// TIA Portal V17 export
// export: Created 2025-03-05T08:03:03.6083882Z, ExportSetting WithDefaults, DisplayName Totally Integrated Automation Portal, DisplayVersion V17 Update 8, DisplayName TIA Portal Openness, DisplayVersion V17 Update 8, DisplayName TIA Portal Version Control Interface, DisplayVersion V17, DisplayName SINAMICS Startdrive Advanced, DisplayVersion V17 SP2, DisplayName SINAMICS Startdrive G110M, G120, G120C, G120D, G120P, G115D, DisplayVersion V17 SP2, DisplayName SINAMICS Startdrive G130, G150, S120, S150, SINAMICS MV, S210, DisplayVersion V17 SP2, DisplayName STEP 7 Professional, DisplayVersion V17 Update 8, DisplayName SINUMERIK ONE STEP 7 Toolbox, DisplayVersion V17 Update 12, DisplayName SINUMERIK 840D sl STEP 7 Toolbox, DisplayVersion V17 Update 12, DisplayName STEP 7 Safety, DisplayVersion V17 Update 6, DisplayName WinCC Advanced, DisplayVersion V17 Update 8
FUNCTION_BLOCK "FB21014_POWDER_FEEDER_PROFINET"   // FB21014, LAD
TITLE = FB21014 POWDER FEEDER PROFINET
{ S7_Optimized_Access := 'FALSE' }
VERSION : 0.1
// stored: AutoNumber false, IsIECCheckEnabled false, SetENOAutomatically false, UDAEnableTagReadback false
   VAR_INPUT
      "iHMI_Values Setpoints" : "POWDER FEEDER HMI VALUES SETPOINTS";
      "iHMI_Offsets Alarms and Warnings" : "POWDER FEEDER HMI OFFSETS ALARMS WARNINGS";
      "iCNC_Values Setpoints" : "POWDER FEEDER CNC VALUES SETPOINTS";
      iSTOP_LINE_1_VALUES_SETPOINTS : Struct
         LINE_1_GAS_FLOW : Real;   // LINE 1 GAS FLOW SETPOINT
         LINE_1_DISK_SPEED : Real;   // LINE 1 DISK SPEED SETPOINT
      END_STRUCT;
      iSTOP_LINE_2_VALUES_SETPOINTS : Struct
         LINE_2_GAS_FLOW : Real;   // LINE 2 GAS FLOW SETPOINT
         LINE_2_DISK_SPEED : Real;   // LINE 2 DISK SPEED SETPOINT
      END_STRUCT;
      iSTART_LINE_1_VALUES_SETPOINTS : Struct
         LINE_1_GAS_FLOW : Real;   // LINE 1 GAS FLOW SETPOINT
         LINE_1_DISK_SPEED : Real;   // LINE 1 DISK SPEED SETPOINT
      END_STRUCT;
      iSTART_LINE_2_VALUES_SETPOINTS : Struct
         LINE_2_GAS_FLOW : Real;   // LINE 2 GAS FLOW SETPOINT
         LINE_2_DISK_SPEED : Real;   // LINE 2 DISK SPEED SETPOINT
      END_STRUCT;
      iArgon_Carrier_Gas_Selected : Bool;
      iNitro_Carrier_Gas_Selected : Bool;
      iHelium_Carrier_Gas_Selected : Bool;
      iArgon30_Carrier_Gas_Selected : Bool;
      iLINE_1_ON_SEQ_ON : Bool;
      iLINE_2_ON_SEQ_ON : Bool;
      iLINE_1_OFF_SEQ_ON : Bool;
      iLINE_2_OFF_SEQ_ON : Bool;
      iLINE_1_STOPPED : Bool;   // HOPPER LINE 1 STOPPPED
      iLINE_2_STOPPED : Bool;   // HOPPER LINE 2 STOPPPED
   END_VAR
   VAR_OUTPUT
      oPLC_Aux : "POWDER FEEDER PLC AUXILIAR";
      oSTATION_WARNINGS : Bool;
      oWARNING_PF_LINE_1_GRAVIMETRIC_MODE_SELECTED : Bool;
      oWARNING_PF_LINE_2_GRAVIMETRIC_MODE_SELECTED : Bool;
   END_VAR
   VAR_IN_OUT
      ioPowder_Feeder_Unit_In_Out : "POWDER FEEDER OERLIKON";
   END_VAR
   VAR DB_SPECIFIC
      INPUT_SETTINGS : Struct
         UNIT_NUMBER : Int;
         FEEDER_NUMBER : Int;
      END_STRUCT;
      AUX_MANUAL_GAS_LINE_1 : Bool;   // AUX MANUAL GAS LINE 1
      AUX_MANUAL_GAS_LINE_2 : Bool;   // AUX MANUAL GAS LINE 2
      AUX_MANUAL_DISK_LINE_1 : Bool;   // AUX MANUAL DISK LINE 1
      AUX_MANUAL_DISK_LINE_2 : Bool;   // AUX MANUAL DISK LINE 2
      swapped : Word;
   END_VAR
   VAR_TEMP
      HMI_INPUT_MAN_MODE : Bool;
      OPTIONS_ON : Bool;
      OPTIONS_OFF : Bool;
      "VOLUMETRIC/GRAVIMETRIC" : Bool;
      "¿SUSTITUIR_VAR_CNC?" : Real;
      Retval_Fill_R : Real;
      DB_NUMBER : DInt;
   END_VAR
   VAR_TEMP   // added for the SCL form of the ladder/FBD networks
      _w1 : Bool;
   END_VAR
BEGIN

NETWORK
TITLE = READ INSTANCE DB NUMBER
      L     DINO;
      +     10#800000;
      T     #DB_NUMBER;

REGION Network 2: HMI INPUT
   // With Hmi Input we allow for user manipulation of feeder operating parameters. If not, they get overriden by robot interlock.
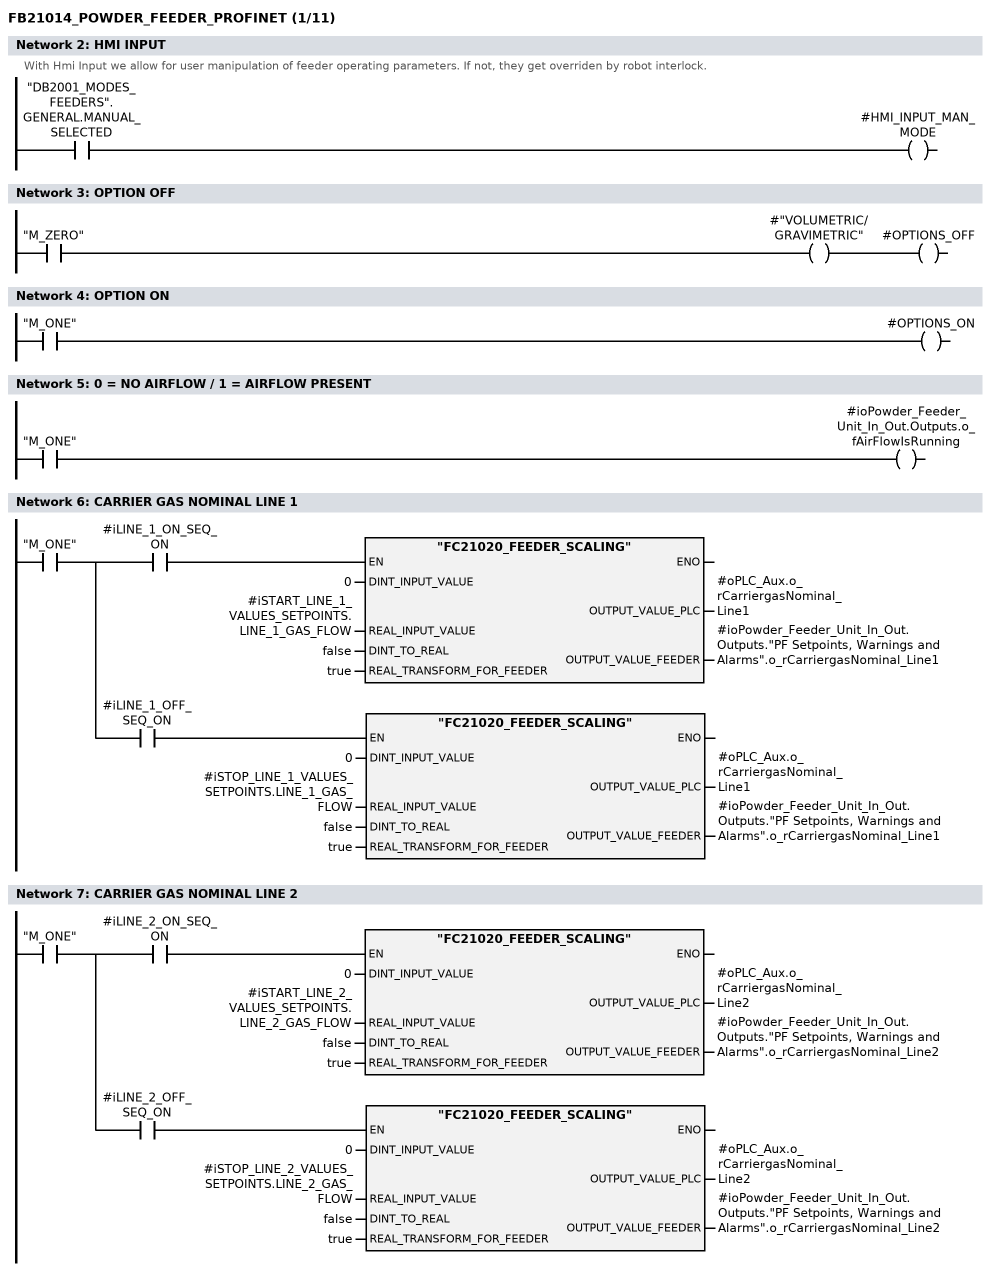
   RUNG wire#powerrail
      Contact( "DB2001_MODES_FEEDERS".GENERAL.MANUAL_SELECTED )
      Coil( #HMI_INPUT_MAN_MODE )
   END_RUNG
   // the same network as SCL:
   #HMI_INPUT_MAN_MODE := "DB2001_MODES_FEEDERS".GENERAL.MANUAL_SELECTED;
END_REGION

REGION Network 3: OPTION OFF
   RUNG wire#powerrail
      Contact( "M_ZERO" )
      Coil( #"VOLUMETRIC/GRAVIMETRIC" )
      Coil( #OPTIONS_OFF )
   END_RUNG
   // the same network as SCL:
   #"VOLUMETRIC/GRAVIMETRIC" := "M_ZERO";
   #OPTIONS_OFF := "M_ZERO";
END_REGION

REGION Network 4: OPTION ON
   RUNG wire#powerrail
      Contact( "M_ONE" )
      Coil( #OPTIONS_ON )
   END_RUNG
   // the same network as SCL:
   #OPTIONS_ON := "M_ONE";
END_REGION

REGION Network 5: 0 = NO AIRFLOW / 1 = AIRFLOW PRESENT
   RUNG wire#powerrail
      Contact( "M_ONE" )
      Coil( #ioPowder_Feeder_Unit_In_Out.Outputs.o_fAirFlowIsRunning )
   END_RUNG
   // the same network as SCL:
   #ioPowder_Feeder_Unit_In_Out.Outputs.o_fAirFlowIsRunning := "M_ONE";
END_REGION

REGION Network 6: CARRIER GAS NOMINAL LINE 1
   RUNG wire#powerrail
      Contact( "M_ONE" )
      wire#w1
      Contact( #iLINE_1_ON_SEQ_ON )
      "FC21020_FEEDER_SCALING"(DINT_INPUT_VALUE := 0, REAL_INPUT_VALUE := #iSTART_LINE_1_VALUES_SETPOINTS.LINE_1_GAS_FLOW, DINT_TO_REAL := false, REAL_TRANSFORM_FOR_FEEDER := true, OUTPUT_VALUE_PLC => #oPLC_Aux.o_rCarriergasNominal_Line1, OUTPUT_VALUE_FEEDER => #ioPowder_Feeder_Unit_In_Out.Outputs."PF Setpoints, Warnings and Alarms".o_rCarriergasNominal_Line1)
   END_RUNG
   RUNG wire#w1
      Contact( #iLINE_1_OFF_SEQ_ON )
      "FC21020_FEEDER_SCALING"(DINT_INPUT_VALUE := 0, REAL_INPUT_VALUE := #iSTOP_LINE_1_VALUES_SETPOINTS.LINE_1_GAS_FLOW, DINT_TO_REAL := false, REAL_TRANSFORM_FOR_FEEDER := true, OUTPUT_VALUE_PLC => #oPLC_Aux.o_rCarriergasNominal_Line1, OUTPUT_VALUE_FEEDER => #ioPowder_Feeder_Unit_In_Out.Outputs."PF Setpoints, Warnings and Alarms".o_rCarriergasNominal_Line1)
   END_RUNG
   // the same network as SCL:
   #_w1 := "M_ONE";
   IF "M_ONE" AND #iLINE_1_ON_SEQ_ON THEN
       "FC21020_FEEDER_SCALING"(DINT_INPUT_VALUE := 0,
                               REAL_INPUT_VALUE := #iSTART_LINE_1_VALUES_SETPOINTS.LINE_1_GAS_FLOW,
                               DINT_TO_REAL := false,
                               REAL_TRANSFORM_FOR_FEEDER := true,
                               OUTPUT_VALUE_PLC => #oPLC_Aux.o_rCarriergasNominal_Line1,
                               OUTPUT_VALUE_FEEDER => #ioPowder_Feeder_Unit_In_Out.Outputs."PF Setpoints, Warnings and Alarms".o_rCarriergasNominal_Line1);
   END_IF;
   IF #_w1 AND #iLINE_1_OFF_SEQ_ON THEN
       "FC21020_FEEDER_SCALING"(DINT_INPUT_VALUE := 0,
                               REAL_INPUT_VALUE := #iSTOP_LINE_1_VALUES_SETPOINTS.LINE_1_GAS_FLOW,
                               DINT_TO_REAL := false,
                               REAL_TRANSFORM_FOR_FEEDER := true,
                               OUTPUT_VALUE_PLC => #oPLC_Aux.o_rCarriergasNominal_Line1,
                               OUTPUT_VALUE_FEEDER => #ioPowder_Feeder_Unit_In_Out.Outputs."PF Setpoints, Warnings and Alarms".o_rCarriergasNominal_Line1);
   END_IF;
END_REGION

REGION Network 7: CARRIER GAS NOMINAL LINE 2
   RUNG wire#powerrail
      Contact( "M_ONE" )
      wire#w1
      Contact( #iLINE_2_ON_SEQ_ON )
      "FC21020_FEEDER_SCALING"(DINT_INPUT_VALUE := 0, REAL_INPUT_VALUE := #iSTART_LINE_2_VALUES_SETPOINTS.LINE_2_GAS_FLOW, DINT_TO_REAL := false, REAL_TRANSFORM_FOR_FEEDER := true, OUTPUT_VALUE_PLC => #oPLC_Aux.o_rCarriergasNominal_Line2, OUTPUT_VALUE_FEEDER => #ioPowder_Feeder_Unit_In_Out.Outputs."PF Setpoints, Warnings and Alarms".o_rCarriergasNominal_Line2)
   END_RUNG
   RUNG wire#w1
      Contact( #iLINE_2_OFF_SEQ_ON )
      "FC21020_FEEDER_SCALING"(DINT_INPUT_VALUE := 0, REAL_INPUT_VALUE := #iSTOP_LINE_2_VALUES_SETPOINTS.LINE_2_GAS_FLOW, DINT_TO_REAL := false, REAL_TRANSFORM_FOR_FEEDER := true, OUTPUT_VALUE_PLC => #oPLC_Aux.o_rCarriergasNominal_Line2, OUTPUT_VALUE_FEEDER => #ioPowder_Feeder_Unit_In_Out.Outputs."PF Setpoints, Warnings and Alarms".o_rCarriergasNominal_Line2)
   END_RUNG
   // the same network as SCL:
   #_w1 := "M_ONE";
   IF "M_ONE" AND #iLINE_2_ON_SEQ_ON THEN
       "FC21020_FEEDER_SCALING"(DINT_INPUT_VALUE := 0,
                               REAL_INPUT_VALUE := #iSTART_LINE_2_VALUES_SETPOINTS.LINE_2_GAS_FLOW,
                               DINT_TO_REAL := false,
                               REAL_TRANSFORM_FOR_FEEDER := true,
                               OUTPUT_VALUE_PLC => #oPLC_Aux.o_rCarriergasNominal_Line2,
                               OUTPUT_VALUE_FEEDER => #ioPowder_Feeder_Unit_In_Out.Outputs."PF Setpoints, Warnings and Alarms".o_rCarriergasNominal_Line2);
   END_IF;
   IF #_w1 AND #iLINE_2_OFF_SEQ_ON THEN
       "FC21020_FEEDER_SCALING"(DINT_INPUT_VALUE := 0,
                               REAL_INPUT_VALUE := #iSTOP_LINE_2_VALUES_SETPOINTS.LINE_2_GAS_FLOW,
                               DINT_TO_REAL := false,
                               REAL_TRANSFORM_FOR_FEEDER := true,
                               OUTPUT_VALUE_PLC => #oPLC_Aux.o_rCarriergasNominal_Line2,
                               OUTPUT_VALUE_FEEDER => #ioPowder_Feeder_Unit_In_Out.Outputs."PF Setpoints, Warnings and Alarms".o_rCarriergasNominal_Line2);
   END_IF;
END_REGION

REGION Network 8: DISK SPEED NOMINAL LINE 1
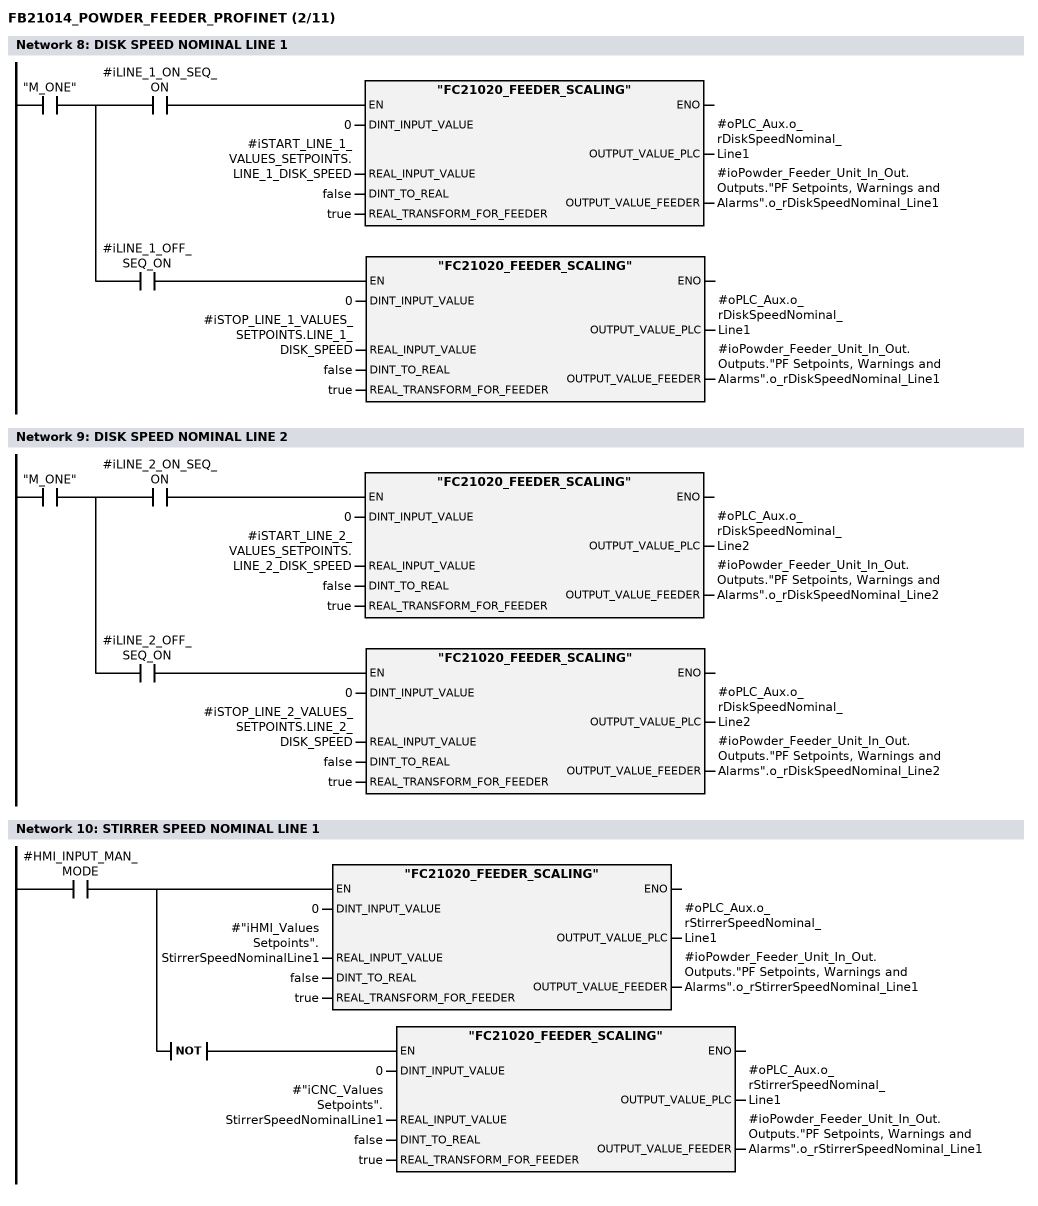
   RUNG wire#powerrail
      Contact( "M_ONE" )
      wire#w1
      Contact( #iLINE_1_ON_SEQ_ON )
      "FC21020_FEEDER_SCALING"(DINT_INPUT_VALUE := 0, REAL_INPUT_VALUE := #iSTART_LINE_1_VALUES_SETPOINTS.LINE_1_DISK_SPEED, DINT_TO_REAL := false, REAL_TRANSFORM_FOR_FEEDER := true, OUTPUT_VALUE_PLC => #oPLC_Aux.o_rDiskSpeedNominal_Line1, OUTPUT_VALUE_FEEDER => #ioPowder_Feeder_Unit_In_Out.Outputs."PF Setpoints, Warnings and Alarms".o_rDiskSpeedNominal_Line1)
   END_RUNG
   RUNG wire#w1
      Contact( #iLINE_1_OFF_SEQ_ON )
      "FC21020_FEEDER_SCALING"(DINT_INPUT_VALUE := 0, REAL_INPUT_VALUE := #iSTOP_LINE_1_VALUES_SETPOINTS.LINE_1_DISK_SPEED, DINT_TO_REAL := false, REAL_TRANSFORM_FOR_FEEDER := true, OUTPUT_VALUE_PLC => #oPLC_Aux.o_rDiskSpeedNominal_Line1, OUTPUT_VALUE_FEEDER => #ioPowder_Feeder_Unit_In_Out.Outputs."PF Setpoints, Warnings and Alarms".o_rDiskSpeedNominal_Line1)
   END_RUNG
   // the same network as SCL:
   #_w1 := "M_ONE";
   IF "M_ONE" AND #iLINE_1_ON_SEQ_ON THEN
       "FC21020_FEEDER_SCALING"(DINT_INPUT_VALUE := 0,
                               REAL_INPUT_VALUE := #iSTART_LINE_1_VALUES_SETPOINTS.LINE_1_DISK_SPEED,
                               DINT_TO_REAL := false,
                               REAL_TRANSFORM_FOR_FEEDER := true,
                               OUTPUT_VALUE_PLC => #oPLC_Aux.o_rDiskSpeedNominal_Line1,
                               OUTPUT_VALUE_FEEDER => #ioPowder_Feeder_Unit_In_Out.Outputs."PF Setpoints, Warnings and Alarms".o_rDiskSpeedNominal_Line1);
   END_IF;
   IF #_w1 AND #iLINE_1_OFF_SEQ_ON THEN
       "FC21020_FEEDER_SCALING"(DINT_INPUT_VALUE := 0,
                               REAL_INPUT_VALUE := #iSTOP_LINE_1_VALUES_SETPOINTS.LINE_1_DISK_SPEED,
                               DINT_TO_REAL := false,
                               REAL_TRANSFORM_FOR_FEEDER := true,
                               OUTPUT_VALUE_PLC => #oPLC_Aux.o_rDiskSpeedNominal_Line1,
                               OUTPUT_VALUE_FEEDER => #ioPowder_Feeder_Unit_In_Out.Outputs."PF Setpoints, Warnings and Alarms".o_rDiskSpeedNominal_Line1);
   END_IF;
END_REGION

REGION Network 9: DISK SPEED NOMINAL LINE 2
   RUNG wire#powerrail
      Contact( "M_ONE" )
      wire#w1
      Contact( #iLINE_2_ON_SEQ_ON )
      "FC21020_FEEDER_SCALING"(DINT_INPUT_VALUE := 0, REAL_INPUT_VALUE := #iSTART_LINE_2_VALUES_SETPOINTS.LINE_2_DISK_SPEED, DINT_TO_REAL := false, REAL_TRANSFORM_FOR_FEEDER := true, OUTPUT_VALUE_PLC => #oPLC_Aux.o_rDiskSpeedNominal_Line2, OUTPUT_VALUE_FEEDER => #ioPowder_Feeder_Unit_In_Out.Outputs."PF Setpoints, Warnings and Alarms".o_rDiskSpeedNominal_Line2)
   END_RUNG
   RUNG wire#w1
      Contact( #iLINE_2_OFF_SEQ_ON )
      "FC21020_FEEDER_SCALING"(DINT_INPUT_VALUE := 0, REAL_INPUT_VALUE := #iSTOP_LINE_2_VALUES_SETPOINTS.LINE_2_DISK_SPEED, DINT_TO_REAL := false, REAL_TRANSFORM_FOR_FEEDER := true, OUTPUT_VALUE_PLC => #oPLC_Aux.o_rDiskSpeedNominal_Line2, OUTPUT_VALUE_FEEDER => #ioPowder_Feeder_Unit_In_Out.Outputs."PF Setpoints, Warnings and Alarms".o_rDiskSpeedNominal_Line2)
   END_RUNG
   // the same network as SCL:
   #_w1 := "M_ONE";
   IF "M_ONE" AND #iLINE_2_ON_SEQ_ON THEN
       "FC21020_FEEDER_SCALING"(DINT_INPUT_VALUE := 0,
                               REAL_INPUT_VALUE := #iSTART_LINE_2_VALUES_SETPOINTS.LINE_2_DISK_SPEED,
                               DINT_TO_REAL := false,
                               REAL_TRANSFORM_FOR_FEEDER := true,
                               OUTPUT_VALUE_PLC => #oPLC_Aux.o_rDiskSpeedNominal_Line2,
                               OUTPUT_VALUE_FEEDER => #ioPowder_Feeder_Unit_In_Out.Outputs."PF Setpoints, Warnings and Alarms".o_rDiskSpeedNominal_Line2);
   END_IF;
   IF #_w1 AND #iLINE_2_OFF_SEQ_ON THEN
       "FC21020_FEEDER_SCALING"(DINT_INPUT_VALUE := 0,
                               REAL_INPUT_VALUE := #iSTOP_LINE_2_VALUES_SETPOINTS.LINE_2_DISK_SPEED,
                               DINT_TO_REAL := false,
                               REAL_TRANSFORM_FOR_FEEDER := true,
                               OUTPUT_VALUE_PLC => #oPLC_Aux.o_rDiskSpeedNominal_Line2,
                               OUTPUT_VALUE_FEEDER => #ioPowder_Feeder_Unit_In_Out.Outputs."PF Setpoints, Warnings and Alarms".o_rDiskSpeedNominal_Line2);
   END_IF;
END_REGION

REGION Network 10: STIRRER SPEED NOMINAL LINE 1
   RUNG wire#powerrail
      Contact( #HMI_INPUT_MAN_MODE )
      wire#w1
      "FC21020_FEEDER_SCALING"(DINT_INPUT_VALUE := 0, REAL_INPUT_VALUE := #"iHMI_Values Setpoints".StirrerSpeedNominalLine1, DINT_TO_REAL := false, REAL_TRANSFORM_FOR_FEEDER := true, OUTPUT_VALUE_PLC => #oPLC_Aux.o_rStirrerSpeedNominal_Line1, OUTPUT_VALUE_FEEDER => #ioPowder_Feeder_Unit_In_Out.Outputs."PF Setpoints, Warnings and Alarms".o_rStirrerSpeedNominal_Line1)
   END_RUNG
   RUNG wire#w1
      Not()
      "FC21020_FEEDER_SCALING"(DINT_INPUT_VALUE := 0, REAL_INPUT_VALUE := #"iCNC_Values Setpoints".StirrerSpeedNominalLine1, DINT_TO_REAL := false, REAL_TRANSFORM_FOR_FEEDER := true, OUTPUT_VALUE_PLC => #oPLC_Aux.o_rStirrerSpeedNominal_Line1, OUTPUT_VALUE_FEEDER => #ioPowder_Feeder_Unit_In_Out.Outputs."PF Setpoints, Warnings and Alarms".o_rStirrerSpeedNominal_Line1)
   END_RUNG
   // the same network as SCL:
   IF #HMI_INPUT_MAN_MODE THEN
       "FC21020_FEEDER_SCALING"(DINT_INPUT_VALUE := 0,
                               REAL_INPUT_VALUE := #"iHMI_Values Setpoints".StirrerSpeedNominalLine1,
                               DINT_TO_REAL := false,
                               REAL_TRANSFORM_FOR_FEEDER := true,
                               OUTPUT_VALUE_PLC => #oPLC_Aux.o_rStirrerSpeedNominal_Line1,
                               OUTPUT_VALUE_FEEDER => #ioPowder_Feeder_Unit_In_Out.Outputs."PF Setpoints, Warnings and Alarms".o_rStirrerSpeedNominal_Line1);
   END_IF;
   IF NOT #HMI_INPUT_MAN_MODE THEN
       "FC21020_FEEDER_SCALING"(DINT_INPUT_VALUE := 0,
                               REAL_INPUT_VALUE := #"iCNC_Values Setpoints".StirrerSpeedNominalLine1,
                               DINT_TO_REAL := false,
                               REAL_TRANSFORM_FOR_FEEDER := true,
                               OUTPUT_VALUE_PLC => #oPLC_Aux.o_rStirrerSpeedNominal_Line1,
                               OUTPUT_VALUE_FEEDER => #ioPowder_Feeder_Unit_In_Out.Outputs."PF Setpoints, Warnings and Alarms".o_rStirrerSpeedNominal_Line1);
   END_IF;
END_REGION

REGION Network 11: STIRRER SPEED NOMINAL LINE 2
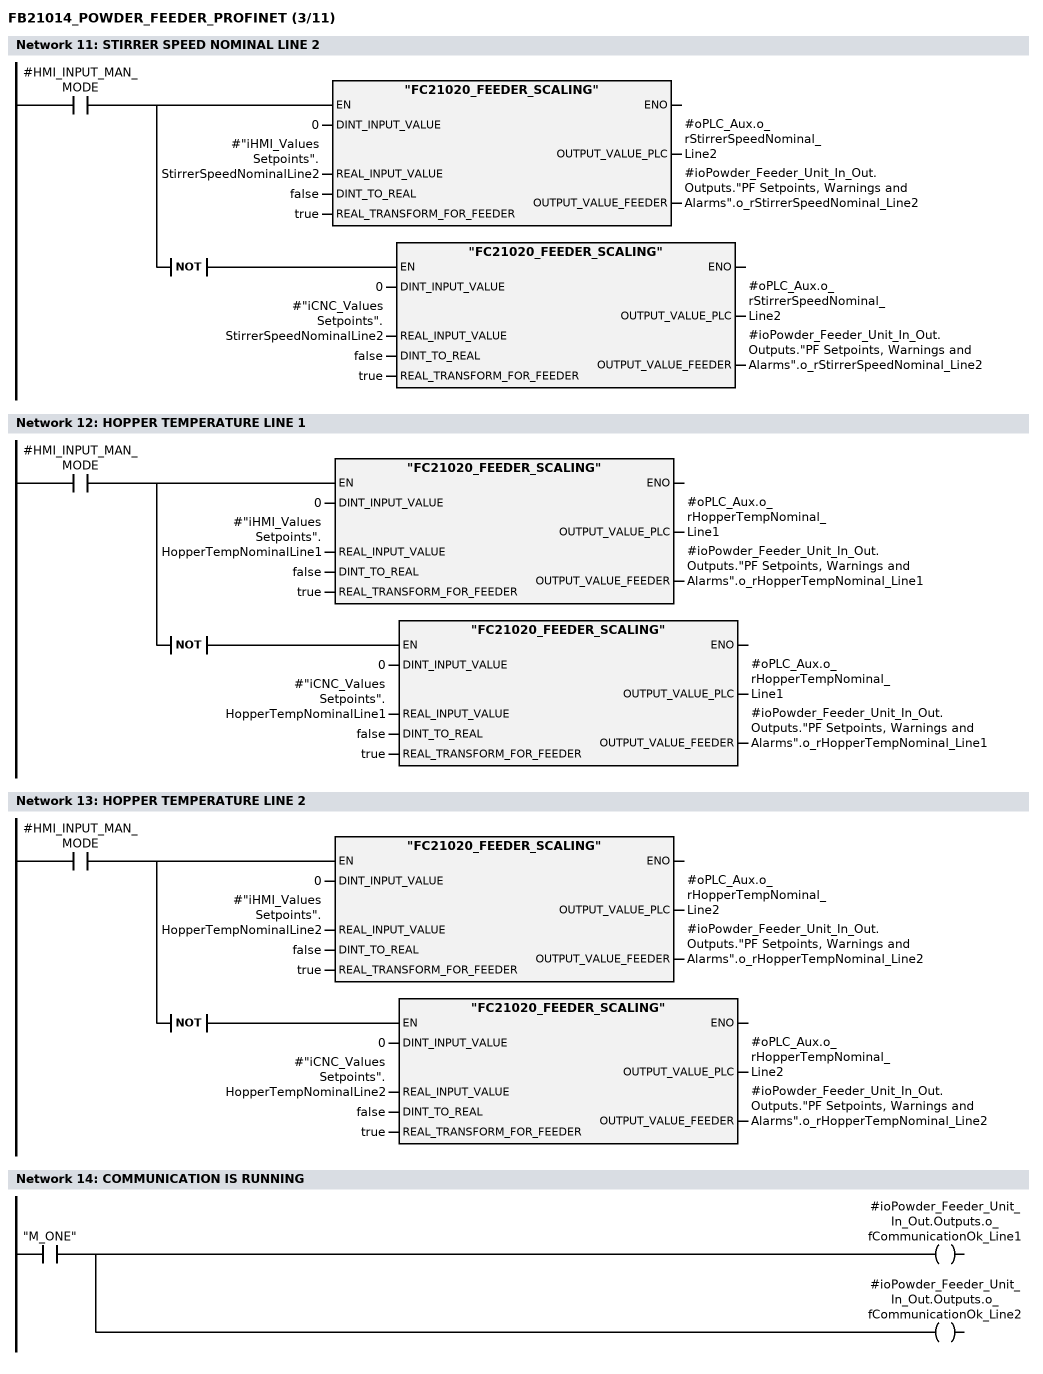
   RUNG wire#powerrail
      Contact( #HMI_INPUT_MAN_MODE )
      wire#w1
      "FC21020_FEEDER_SCALING"(DINT_INPUT_VALUE := 0, REAL_INPUT_VALUE := #"iHMI_Values Setpoints".StirrerSpeedNominalLine2, DINT_TO_REAL := false, REAL_TRANSFORM_FOR_FEEDER := true, OUTPUT_VALUE_PLC => #oPLC_Aux.o_rStirrerSpeedNominal_Line2, OUTPUT_VALUE_FEEDER => #ioPowder_Feeder_Unit_In_Out.Outputs."PF Setpoints, Warnings and Alarms".o_rStirrerSpeedNominal_Line2)
   END_RUNG
   RUNG wire#w1
      Not()
      "FC21020_FEEDER_SCALING"(DINT_INPUT_VALUE := 0, REAL_INPUT_VALUE := #"iCNC_Values Setpoints".StirrerSpeedNominalLine2, DINT_TO_REAL := false, REAL_TRANSFORM_FOR_FEEDER := true, OUTPUT_VALUE_PLC => #oPLC_Aux.o_rStirrerSpeedNominal_Line2, OUTPUT_VALUE_FEEDER => #ioPowder_Feeder_Unit_In_Out.Outputs."PF Setpoints, Warnings and Alarms".o_rStirrerSpeedNominal_Line2)
   END_RUNG
   // the same network as SCL:
   IF #HMI_INPUT_MAN_MODE THEN
       "FC21020_FEEDER_SCALING"(DINT_INPUT_VALUE := 0,
                               REAL_INPUT_VALUE := #"iHMI_Values Setpoints".StirrerSpeedNominalLine2,
                               DINT_TO_REAL := false,
                               REAL_TRANSFORM_FOR_FEEDER := true,
                               OUTPUT_VALUE_PLC => #oPLC_Aux.o_rStirrerSpeedNominal_Line2,
                               OUTPUT_VALUE_FEEDER => #ioPowder_Feeder_Unit_In_Out.Outputs."PF Setpoints, Warnings and Alarms".o_rStirrerSpeedNominal_Line2);
   END_IF;
   IF NOT #HMI_INPUT_MAN_MODE THEN
       "FC21020_FEEDER_SCALING"(DINT_INPUT_VALUE := 0,
                               REAL_INPUT_VALUE := #"iCNC_Values Setpoints".StirrerSpeedNominalLine2,
                               DINT_TO_REAL := false,
                               REAL_TRANSFORM_FOR_FEEDER := true,
                               OUTPUT_VALUE_PLC => #oPLC_Aux.o_rStirrerSpeedNominal_Line2,
                               OUTPUT_VALUE_FEEDER => #ioPowder_Feeder_Unit_In_Out.Outputs."PF Setpoints, Warnings and Alarms".o_rStirrerSpeedNominal_Line2);
   END_IF;
END_REGION

REGION Network 12: HOPPER TEMPERATURE LINE 1
   RUNG wire#powerrail
      Contact( #HMI_INPUT_MAN_MODE )
      wire#w1
      "FC21020_FEEDER_SCALING"(DINT_INPUT_VALUE := 0, REAL_INPUT_VALUE := #"iHMI_Values Setpoints".HopperTempNominalLine1, DINT_TO_REAL := false, REAL_TRANSFORM_FOR_FEEDER := true, OUTPUT_VALUE_PLC => #oPLC_Aux.o_rHopperTempNominal_Line1, OUTPUT_VALUE_FEEDER => #ioPowder_Feeder_Unit_In_Out.Outputs."PF Setpoints, Warnings and Alarms".o_rHopperTempNominal_Line1)
   END_RUNG
   RUNG wire#w1
      Not()
      "FC21020_FEEDER_SCALING"(DINT_INPUT_VALUE := 0, REAL_INPUT_VALUE := #"iCNC_Values Setpoints".HopperTempNominalLine1, DINT_TO_REAL := false, REAL_TRANSFORM_FOR_FEEDER := true, OUTPUT_VALUE_PLC => #oPLC_Aux.o_rHopperTempNominal_Line1, OUTPUT_VALUE_FEEDER => #ioPowder_Feeder_Unit_In_Out.Outputs."PF Setpoints, Warnings and Alarms".o_rHopperTempNominal_Line1)
   END_RUNG
   // the same network as SCL:
   IF #HMI_INPUT_MAN_MODE THEN
       "FC21020_FEEDER_SCALING"(DINT_INPUT_VALUE := 0,
                               REAL_INPUT_VALUE := #"iHMI_Values Setpoints".HopperTempNominalLine1,
                               DINT_TO_REAL := false,
                               REAL_TRANSFORM_FOR_FEEDER := true,
                               OUTPUT_VALUE_PLC => #oPLC_Aux.o_rHopperTempNominal_Line1,
                               OUTPUT_VALUE_FEEDER => #ioPowder_Feeder_Unit_In_Out.Outputs."PF Setpoints, Warnings and Alarms".o_rHopperTempNominal_Line1);
   END_IF;
   IF NOT #HMI_INPUT_MAN_MODE THEN
       "FC21020_FEEDER_SCALING"(DINT_INPUT_VALUE := 0,
                               REAL_INPUT_VALUE := #"iCNC_Values Setpoints".HopperTempNominalLine1,
                               DINT_TO_REAL := false,
                               REAL_TRANSFORM_FOR_FEEDER := true,
                               OUTPUT_VALUE_PLC => #oPLC_Aux.o_rHopperTempNominal_Line1,
                               OUTPUT_VALUE_FEEDER => #ioPowder_Feeder_Unit_In_Out.Outputs."PF Setpoints, Warnings and Alarms".o_rHopperTempNominal_Line1);
   END_IF;
END_REGION

REGION Network 13: HOPPER TEMPERATURE LINE 2
   RUNG wire#powerrail
      Contact( #HMI_INPUT_MAN_MODE )
      wire#w1
      "FC21020_FEEDER_SCALING"(DINT_INPUT_VALUE := 0, REAL_INPUT_VALUE := #"iHMI_Values Setpoints".HopperTempNominalLine2, DINT_TO_REAL := false, REAL_TRANSFORM_FOR_FEEDER := true, OUTPUT_VALUE_PLC => #oPLC_Aux.o_rHopperTempNominal_Line2, OUTPUT_VALUE_FEEDER => #ioPowder_Feeder_Unit_In_Out.Outputs."PF Setpoints, Warnings and Alarms".o_rHopperTempNominal_Line2)
   END_RUNG
   RUNG wire#w1
      Not()
      "FC21020_FEEDER_SCALING"(DINT_INPUT_VALUE := 0, REAL_INPUT_VALUE := #"iCNC_Values Setpoints".HopperTempNominalLine2, DINT_TO_REAL := false, REAL_TRANSFORM_FOR_FEEDER := true, OUTPUT_VALUE_PLC => #oPLC_Aux.o_rHopperTempNominal_Line2, OUTPUT_VALUE_FEEDER => #ioPowder_Feeder_Unit_In_Out.Outputs."PF Setpoints, Warnings and Alarms".o_rHopperTempNominal_Line2)
   END_RUNG
   // the same network as SCL:
   IF #HMI_INPUT_MAN_MODE THEN
       "FC21020_FEEDER_SCALING"(DINT_INPUT_VALUE := 0,
                               REAL_INPUT_VALUE := #"iHMI_Values Setpoints".HopperTempNominalLine2,
                               DINT_TO_REAL := false,
                               REAL_TRANSFORM_FOR_FEEDER := true,
                               OUTPUT_VALUE_PLC => #oPLC_Aux.o_rHopperTempNominal_Line2,
                               OUTPUT_VALUE_FEEDER => #ioPowder_Feeder_Unit_In_Out.Outputs."PF Setpoints, Warnings and Alarms".o_rHopperTempNominal_Line2);
   END_IF;
   IF NOT #HMI_INPUT_MAN_MODE THEN
       "FC21020_FEEDER_SCALING"(DINT_INPUT_VALUE := 0,
                               REAL_INPUT_VALUE := #"iCNC_Values Setpoints".HopperTempNominalLine2,
                               DINT_TO_REAL := false,
                               REAL_TRANSFORM_FOR_FEEDER := true,
                               OUTPUT_VALUE_PLC => #oPLC_Aux.o_rHopperTempNominal_Line2,
                               OUTPUT_VALUE_FEEDER => #ioPowder_Feeder_Unit_In_Out.Outputs."PF Setpoints, Warnings and Alarms".o_rHopperTempNominal_Line2);
   END_IF;
END_REGION

REGION Network 14: COMMUNICATION IS RUNNING
   RUNG wire#powerrail
      Contact( "M_ONE" )
      wire#w1
      Coil( #ioPowder_Feeder_Unit_In_Out.Outputs.o_fCommunicationOk_Line1 )
   END_RUNG
   RUNG wire#w1
      Coil( #ioPowder_Feeder_Unit_In_Out.Outputs.o_fCommunicationOk_Line2 )
   END_RUNG
   // the same network as SCL:
   #ioPowder_Feeder_Unit_In_Out.Outputs.o_fCommunicationOk_Line1 := "M_ONE";
   #ioPowder_Feeder_Unit_In_Out.Outputs.o_fCommunicationOk_Line2 := "M_ONE";
END_REGION

REGION Network 15: VOLUMETRIC MODE ON
   // Volumetric Mode On = 1 for Twin 150
   // Gravimetric Mode - n/a for Twin 150
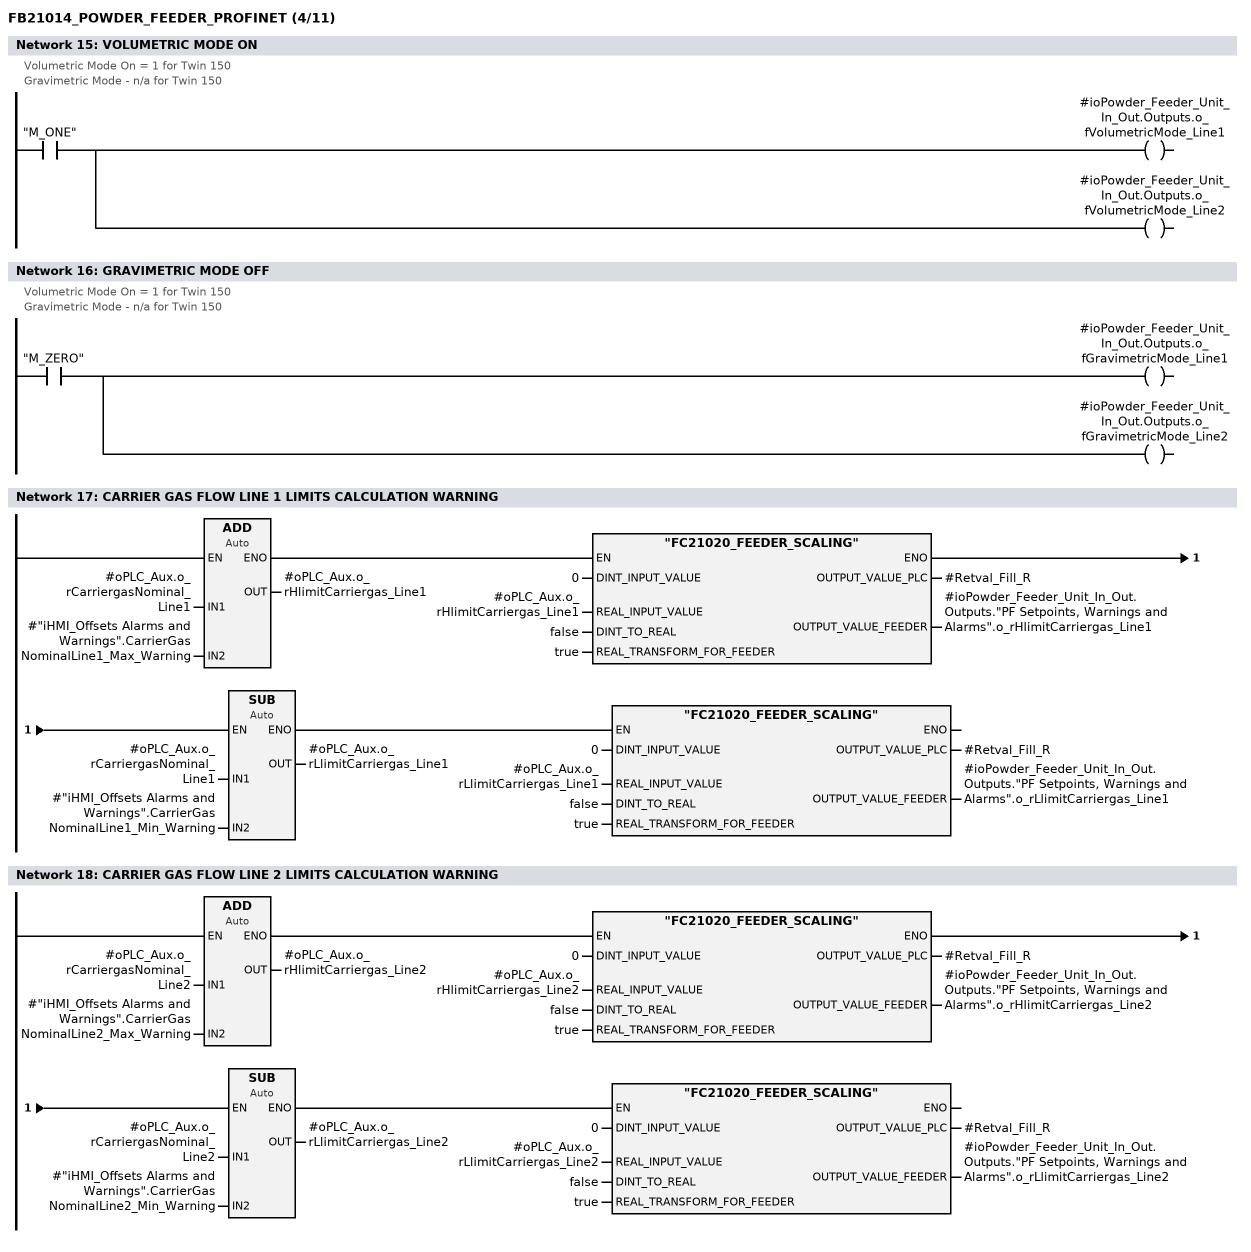
   RUNG wire#powerrail
      Contact( "M_ONE" )
      wire#w1
      Coil( #ioPowder_Feeder_Unit_In_Out.Outputs.o_fVolumetricMode_Line1 )
   END_RUNG
   RUNG wire#w1
      Coil( #ioPowder_Feeder_Unit_In_Out.Outputs.o_fVolumetricMode_Line2 )
   END_RUNG
   // the same network as SCL:
   #ioPowder_Feeder_Unit_In_Out.Outputs.o_fVolumetricMode_Line1 := "M_ONE";
   #ioPowder_Feeder_Unit_In_Out.Outputs.o_fVolumetricMode_Line2 := "M_ONE";
END_REGION

REGION Network 16: GRAVIMETRIC MODE OFF
   // Volumetric Mode On = 1 for Twin 150
   // Gravimetric Mode - n/a for Twin 150
   RUNG wire#powerrail
      Contact( "M_ZERO" )
      wire#w1
      Coil( #ioPowder_Feeder_Unit_In_Out.Outputs.o_fGravimetricMode_Line1 )
   END_RUNG
   RUNG wire#w1
      Coil( #ioPowder_Feeder_Unit_In_Out.Outputs.o_fGravimetricMode_Line2 )
   END_RUNG
   // the same network as SCL:
   #ioPowder_Feeder_Unit_In_Out.Outputs.o_fGravimetricMode_Line1 := "M_ZERO";
   #ioPowder_Feeder_Unit_In_Out.Outputs.o_fGravimetricMode_Line2 := "M_ZERO";
END_REGION

REGION Network 17: CARRIER GAS FLOW LINE 1 LIMITS CALCULATION WARNING
   RUNG wire#powerrail
      Add(in1 := #oPLC_Aux.o_rCarriergasNominal_Line1, in2 := #"iHMI_Offsets Alarms and Warnings".CarrierGasNominalLine1_Max_Warning, out => #oPLC_Aux.o_rHlimitCarriergas_Line1)
      "FC21020_FEEDER_SCALING"(DINT_INPUT_VALUE := 0, REAL_INPUT_VALUE := #oPLC_Aux.o_rHlimitCarriergas_Line1, DINT_TO_REAL := false, REAL_TRANSFORM_FOR_FEEDER := true, OUTPUT_VALUE_PLC => #Retval_Fill_R, OUTPUT_VALUE_FEEDER => #ioPowder_Feeder_Unit_In_Out.Outputs."PF Setpoints, Warnings and Alarms".o_rHlimitCarriergas_Line1)
      Sub(in1 := #oPLC_Aux.o_rCarriergasNominal_Line1, in2 := #"iHMI_Offsets Alarms and Warnings".CarrierGasNominalLine1_Min_Warning, out => #oPLC_Aux.o_rLlimitCarriergas_Line1)
      "FC21020_FEEDER_SCALING"(DINT_INPUT_VALUE := 0, REAL_INPUT_VALUE := #oPLC_Aux.o_rLlimitCarriergas_Line1, DINT_TO_REAL := false, REAL_TRANSFORM_FOR_FEEDER := true, OUTPUT_VALUE_PLC => #Retval_Fill_R, OUTPUT_VALUE_FEEDER => #ioPowder_Feeder_Unit_In_Out.Outputs."PF Setpoints, Warnings and Alarms".o_rLlimitCarriergas_Line1)
   END_RUNG
   // the same network as SCL:
   #oPLC_Aux.o_rHlimitCarriergas_Line1 := #oPLC_Aux.o_rCarriergasNominal_Line1 + #"iHMI_Offsets Alarms and Warnings".CarrierGasNominalLine1_Max_Warning;
   "FC21020_FEEDER_SCALING"(DINT_INPUT_VALUE := 0,
                           REAL_INPUT_VALUE := #oPLC_Aux.o_rHlimitCarriergas_Line1,
                           DINT_TO_REAL := false,
                           REAL_TRANSFORM_FOR_FEEDER := true,
                           OUTPUT_VALUE_PLC => #Retval_Fill_R,
                           OUTPUT_VALUE_FEEDER => #ioPowder_Feeder_Unit_In_Out.Outputs."PF Setpoints, Warnings and Alarms".o_rHlimitCarriergas_Line1,
                           ENO => #_w1);
   IF #_w1 THEN
       #oPLC_Aux.o_rLlimitCarriergas_Line1 := #oPLC_Aux.o_rCarriergasNominal_Line1 - #"iHMI_Offsets Alarms and Warnings".CarrierGasNominalLine1_Min_Warning;
       "FC21020_FEEDER_SCALING"(DINT_INPUT_VALUE := 0,
                               REAL_INPUT_VALUE := #oPLC_Aux.o_rLlimitCarriergas_Line1,
                               DINT_TO_REAL := false,
                               REAL_TRANSFORM_FOR_FEEDER := true,
                               OUTPUT_VALUE_PLC => #Retval_Fill_R,
                               OUTPUT_VALUE_FEEDER => #ioPowder_Feeder_Unit_In_Out.Outputs."PF Setpoints, Warnings and Alarms".o_rLlimitCarriergas_Line1);
   END_IF;
END_REGION

REGION Network 18: CARRIER GAS FLOW LINE 2 LIMITS CALCULATION WARNING
   RUNG wire#powerrail
      Add(in1 := #oPLC_Aux.o_rCarriergasNominal_Line2, in2 := #"iHMI_Offsets Alarms and Warnings".CarrierGasNominalLine2_Max_Warning, out => #oPLC_Aux.o_rHlimitCarriergas_Line2)
      "FC21020_FEEDER_SCALING"(DINT_INPUT_VALUE := 0, REAL_INPUT_VALUE := #oPLC_Aux.o_rHlimitCarriergas_Line2, DINT_TO_REAL := false, REAL_TRANSFORM_FOR_FEEDER := true, OUTPUT_VALUE_PLC => #Retval_Fill_R, OUTPUT_VALUE_FEEDER => #ioPowder_Feeder_Unit_In_Out.Outputs."PF Setpoints, Warnings and Alarms".o_rHlimitCarriergas_Line2)
      Sub(in1 := #oPLC_Aux.o_rCarriergasNominal_Line2, in2 := #"iHMI_Offsets Alarms and Warnings".CarrierGasNominalLine2_Min_Warning, out => #oPLC_Aux.o_rLlimitCarriergas_Line2)
      "FC21020_FEEDER_SCALING"(DINT_INPUT_VALUE := 0, REAL_INPUT_VALUE := #oPLC_Aux.o_rLlimitCarriergas_Line2, DINT_TO_REAL := false, REAL_TRANSFORM_FOR_FEEDER := true, OUTPUT_VALUE_PLC => #Retval_Fill_R, OUTPUT_VALUE_FEEDER => #ioPowder_Feeder_Unit_In_Out.Outputs."PF Setpoints, Warnings and Alarms".o_rLlimitCarriergas_Line2)
   END_RUNG
   // the same network as SCL:
   #oPLC_Aux.o_rHlimitCarriergas_Line2 := #oPLC_Aux.o_rCarriergasNominal_Line2 + #"iHMI_Offsets Alarms and Warnings".CarrierGasNominalLine2_Max_Warning;
   "FC21020_FEEDER_SCALING"(DINT_INPUT_VALUE := 0,
                           REAL_INPUT_VALUE := #oPLC_Aux.o_rHlimitCarriergas_Line2,
                           DINT_TO_REAL := false,
                           REAL_TRANSFORM_FOR_FEEDER := true,
                           OUTPUT_VALUE_PLC => #Retval_Fill_R,
                           OUTPUT_VALUE_FEEDER => #ioPowder_Feeder_Unit_In_Out.Outputs."PF Setpoints, Warnings and Alarms".o_rHlimitCarriergas_Line2,
                           ENO => #_w1);
   IF #_w1 THEN
       #oPLC_Aux.o_rLlimitCarriergas_Line2 := #oPLC_Aux.o_rCarriergasNominal_Line2 - #"iHMI_Offsets Alarms and Warnings".CarrierGasNominalLine2_Min_Warning;
       "FC21020_FEEDER_SCALING"(DINT_INPUT_VALUE := 0,
                               REAL_INPUT_VALUE := #oPLC_Aux.o_rLlimitCarriergas_Line2,
                               DINT_TO_REAL := false,
                               REAL_TRANSFORM_FOR_FEEDER := true,
                               OUTPUT_VALUE_PLC => #Retval_Fill_R,
                               OUTPUT_VALUE_FEEDER => #ioPowder_Feeder_Unit_In_Out.Outputs."PF Setpoints, Warnings and Alarms".o_rLlimitCarriergas_Line2);
   END_IF;
END_REGION

REGION Network 19: CARRIER GAS FLOW LINE 1 LIMITS CALCULATION ALARM
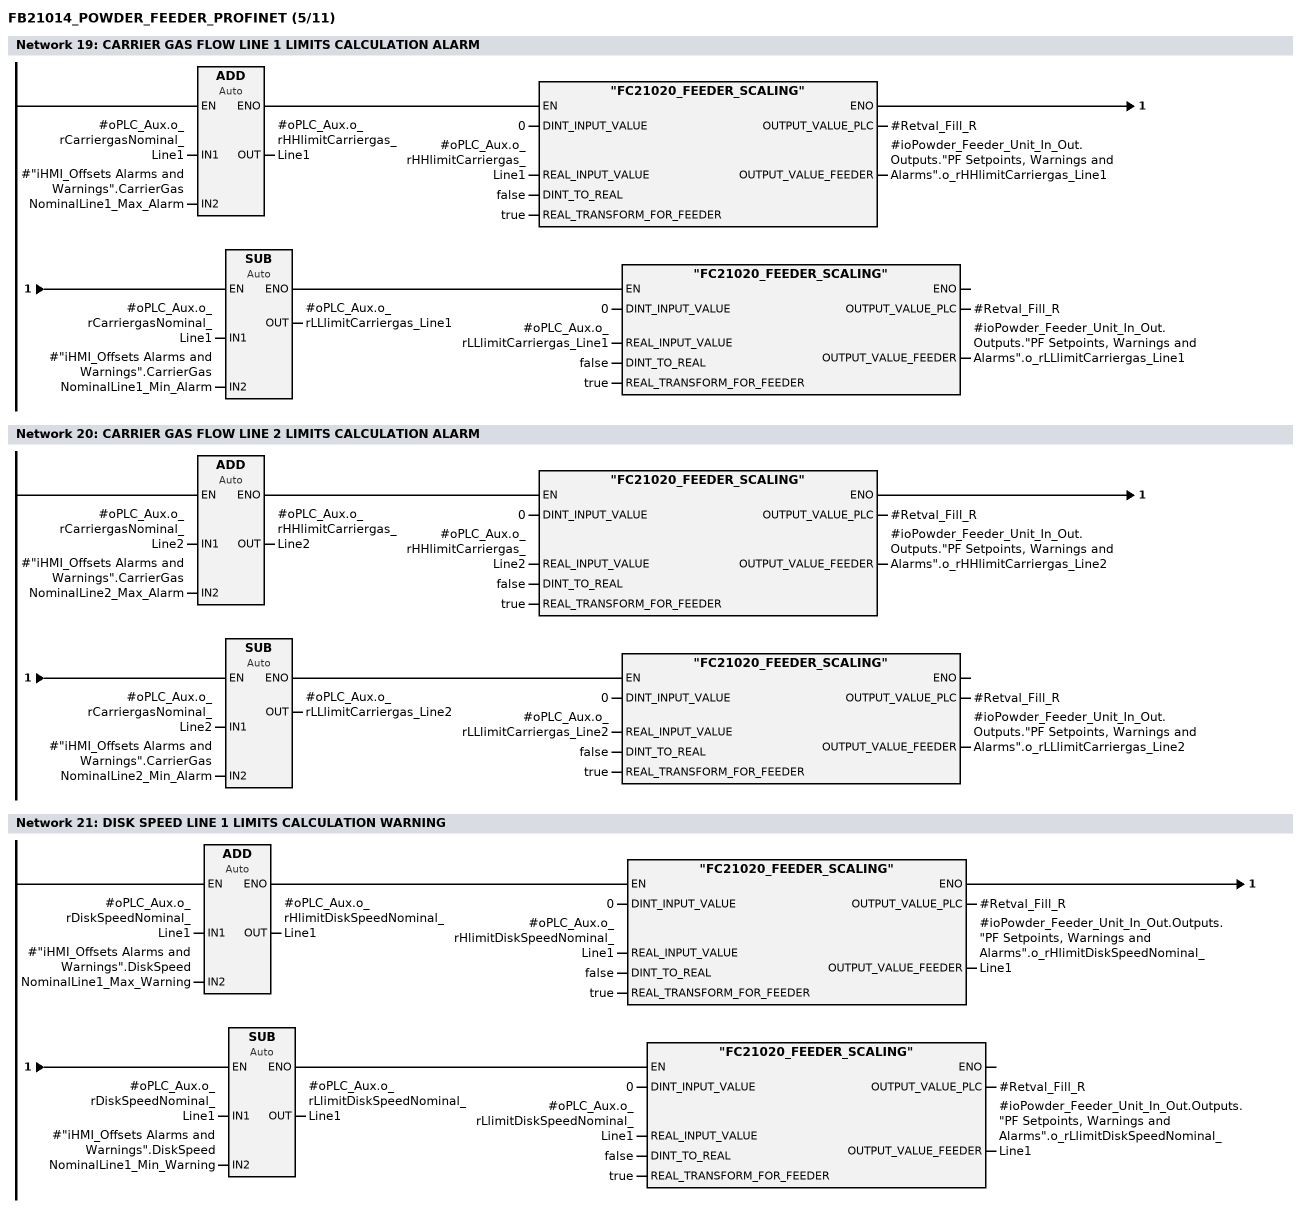
   RUNG wire#powerrail
      Add(in1 := #oPLC_Aux.o_rCarriergasNominal_Line1, in2 := #"iHMI_Offsets Alarms and Warnings".CarrierGasNominalLine1_Max_Alarm, out => #oPLC_Aux.o_rHHlimitCarriergas_Line1)
      "FC21020_FEEDER_SCALING"(DINT_INPUT_VALUE := 0, REAL_INPUT_VALUE := #oPLC_Aux.o_rHHlimitCarriergas_Line1, DINT_TO_REAL := false, REAL_TRANSFORM_FOR_FEEDER := true, OUTPUT_VALUE_PLC => #Retval_Fill_R, OUTPUT_VALUE_FEEDER => #ioPowder_Feeder_Unit_In_Out.Outputs."PF Setpoints, Warnings and Alarms".o_rHHlimitCarriergas_Line1)
      Sub(in1 := #oPLC_Aux.o_rCarriergasNominal_Line1, in2 := #"iHMI_Offsets Alarms and Warnings".CarrierGasNominalLine1_Min_Alarm, out => #oPLC_Aux.o_rLLlimitCarriergas_Line1)
      "FC21020_FEEDER_SCALING"(DINT_INPUT_VALUE := 0, REAL_INPUT_VALUE := #oPLC_Aux.o_rLLlimitCarriergas_Line1, DINT_TO_REAL := false, REAL_TRANSFORM_FOR_FEEDER := true, OUTPUT_VALUE_PLC => #Retval_Fill_R, OUTPUT_VALUE_FEEDER => #ioPowder_Feeder_Unit_In_Out.Outputs."PF Setpoints, Warnings and Alarms".o_rLLlimitCarriergas_Line1)
   END_RUNG
   // the same network as SCL:
   #oPLC_Aux.o_rHHlimitCarriergas_Line1 := #oPLC_Aux.o_rCarriergasNominal_Line1 + #"iHMI_Offsets Alarms and Warnings".CarrierGasNominalLine1_Max_Alarm;
   "FC21020_FEEDER_SCALING"(DINT_INPUT_VALUE := 0,
                           REAL_INPUT_VALUE := #oPLC_Aux.o_rHHlimitCarriergas_Line1,
                           DINT_TO_REAL := false,
                           REAL_TRANSFORM_FOR_FEEDER := true,
                           OUTPUT_VALUE_PLC => #Retval_Fill_R,
                           OUTPUT_VALUE_FEEDER => #ioPowder_Feeder_Unit_In_Out.Outputs."PF Setpoints, Warnings and Alarms".o_rHHlimitCarriergas_Line1,
                           ENO => #_w1);
   IF #_w1 THEN
       #oPLC_Aux.o_rLLlimitCarriergas_Line1 := #oPLC_Aux.o_rCarriergasNominal_Line1 - #"iHMI_Offsets Alarms and Warnings".CarrierGasNominalLine1_Min_Alarm;
       "FC21020_FEEDER_SCALING"(DINT_INPUT_VALUE := 0,
                               REAL_INPUT_VALUE := #oPLC_Aux.o_rLLlimitCarriergas_Line1,
                               DINT_TO_REAL := false,
                               REAL_TRANSFORM_FOR_FEEDER := true,
                               OUTPUT_VALUE_PLC => #Retval_Fill_R,
                               OUTPUT_VALUE_FEEDER => #ioPowder_Feeder_Unit_In_Out.Outputs."PF Setpoints, Warnings and Alarms".o_rLLlimitCarriergas_Line1);
   END_IF;
END_REGION

REGION Network 20: CARRIER GAS FLOW LINE 2 LIMITS CALCULATION ALARM
   RUNG wire#powerrail
      Add(in1 := #oPLC_Aux.o_rCarriergasNominal_Line2, in2 := #"iHMI_Offsets Alarms and Warnings".CarrierGasNominalLine2_Max_Alarm, out => #oPLC_Aux.o_rHHlimitCarriergas_Line2)
      "FC21020_FEEDER_SCALING"(DINT_INPUT_VALUE := 0, REAL_INPUT_VALUE := #oPLC_Aux.o_rHHlimitCarriergas_Line2, DINT_TO_REAL := false, REAL_TRANSFORM_FOR_FEEDER := true, OUTPUT_VALUE_PLC => #Retval_Fill_R, OUTPUT_VALUE_FEEDER => #ioPowder_Feeder_Unit_In_Out.Outputs."PF Setpoints, Warnings and Alarms".o_rHHlimitCarriergas_Line2)
      Sub(in1 := #oPLC_Aux.o_rCarriergasNominal_Line2, in2 := #"iHMI_Offsets Alarms and Warnings".CarrierGasNominalLine2_Min_Alarm, out => #oPLC_Aux.o_rLLlimitCarriergas_Line2)
      "FC21020_FEEDER_SCALING"(DINT_INPUT_VALUE := 0, REAL_INPUT_VALUE := #oPLC_Aux.o_rLLlimitCarriergas_Line2, DINT_TO_REAL := false, REAL_TRANSFORM_FOR_FEEDER := true, OUTPUT_VALUE_PLC => #Retval_Fill_R, OUTPUT_VALUE_FEEDER => #ioPowder_Feeder_Unit_In_Out.Outputs."PF Setpoints, Warnings and Alarms".o_rLLlimitCarriergas_Line2)
   END_RUNG
   // the same network as SCL:
   #oPLC_Aux.o_rHHlimitCarriergas_Line2 := #oPLC_Aux.o_rCarriergasNominal_Line2 + #"iHMI_Offsets Alarms and Warnings".CarrierGasNominalLine2_Max_Alarm;
   "FC21020_FEEDER_SCALING"(DINT_INPUT_VALUE := 0,
                           REAL_INPUT_VALUE := #oPLC_Aux.o_rHHlimitCarriergas_Line2,
                           DINT_TO_REAL := false,
                           REAL_TRANSFORM_FOR_FEEDER := true,
                           OUTPUT_VALUE_PLC => #Retval_Fill_R,
                           OUTPUT_VALUE_FEEDER => #ioPowder_Feeder_Unit_In_Out.Outputs."PF Setpoints, Warnings and Alarms".o_rHHlimitCarriergas_Line2,
                           ENO => #_w1);
   IF #_w1 THEN
       #oPLC_Aux.o_rLLlimitCarriergas_Line2 := #oPLC_Aux.o_rCarriergasNominal_Line2 - #"iHMI_Offsets Alarms and Warnings".CarrierGasNominalLine2_Min_Alarm;
       "FC21020_FEEDER_SCALING"(DINT_INPUT_VALUE := 0,
                               REAL_INPUT_VALUE := #oPLC_Aux.o_rLLlimitCarriergas_Line2,
                               DINT_TO_REAL := false,
                               REAL_TRANSFORM_FOR_FEEDER := true,
                               OUTPUT_VALUE_PLC => #Retval_Fill_R,
                               OUTPUT_VALUE_FEEDER => #ioPowder_Feeder_Unit_In_Out.Outputs."PF Setpoints, Warnings and Alarms".o_rLLlimitCarriergas_Line2);
   END_IF;
END_REGION

REGION Network 21: DISK SPEED LINE 1 LIMITS CALCULATION WARNING
   RUNG wire#powerrail
      Add(in1 := #oPLC_Aux.o_rDiskSpeedNominal_Line1, in2 := #"iHMI_Offsets Alarms and Warnings".DiskSpeedNominalLine1_Max_Warning, out => #oPLC_Aux.o_rHlimitDiskSpeedNominal_Line1)
      "FC21020_FEEDER_SCALING"(DINT_INPUT_VALUE := 0, REAL_INPUT_VALUE := #oPLC_Aux.o_rHlimitDiskSpeedNominal_Line1, DINT_TO_REAL := false, REAL_TRANSFORM_FOR_FEEDER := true, OUTPUT_VALUE_PLC => #Retval_Fill_R, OUTPUT_VALUE_FEEDER => #ioPowder_Feeder_Unit_In_Out.Outputs."PF Setpoints, Warnings and Alarms".o_rHlimitDiskSpeedNominal_Line1)
      Sub(in1 := #oPLC_Aux.o_rDiskSpeedNominal_Line1, in2 := #"iHMI_Offsets Alarms and Warnings".DiskSpeedNominalLine1_Min_Warning, out => #oPLC_Aux.o_rLlimitDiskSpeedNominal_Line1)
      "FC21020_FEEDER_SCALING"(DINT_INPUT_VALUE := 0, REAL_INPUT_VALUE := #oPLC_Aux.o_rLlimitDiskSpeedNominal_Line1, DINT_TO_REAL := false, REAL_TRANSFORM_FOR_FEEDER := true, OUTPUT_VALUE_PLC => #Retval_Fill_R, OUTPUT_VALUE_FEEDER => #ioPowder_Feeder_Unit_In_Out.Outputs."PF Setpoints, Warnings and Alarms".o_rLlimitDiskSpeedNominal_Line1)
   END_RUNG
   // the same network as SCL:
   #oPLC_Aux.o_rHlimitDiskSpeedNominal_Line1 := #oPLC_Aux.o_rDiskSpeedNominal_Line1 + #"iHMI_Offsets Alarms and Warnings".DiskSpeedNominalLine1_Max_Warning;
   "FC21020_FEEDER_SCALING"(DINT_INPUT_VALUE := 0,
                           REAL_INPUT_VALUE := #oPLC_Aux.o_rHlimitDiskSpeedNominal_Line1,
                           DINT_TO_REAL := false,
                           REAL_TRANSFORM_FOR_FEEDER := true,
                           OUTPUT_VALUE_PLC => #Retval_Fill_R,
                           OUTPUT_VALUE_FEEDER => #ioPowder_Feeder_Unit_In_Out.Outputs."PF Setpoints, Warnings and Alarms".o_rHlimitDiskSpeedNominal_Line1,
                           ENO => #_w1);
   IF #_w1 THEN
       #oPLC_Aux.o_rLlimitDiskSpeedNominal_Line1 := #oPLC_Aux.o_rDiskSpeedNominal_Line1 - #"iHMI_Offsets Alarms and Warnings".DiskSpeedNominalLine1_Min_Warning;
       "FC21020_FEEDER_SCALING"(DINT_INPUT_VALUE := 0,
                               REAL_INPUT_VALUE := #oPLC_Aux.o_rLlimitDiskSpeedNominal_Line1,
                               DINT_TO_REAL := false,
                               REAL_TRANSFORM_FOR_FEEDER := true,
                               OUTPUT_VALUE_PLC => #Retval_Fill_R,
                               OUTPUT_VALUE_FEEDER => #ioPowder_Feeder_Unit_In_Out.Outputs."PF Setpoints, Warnings and Alarms".o_rLlimitDiskSpeedNominal_Line1);
   END_IF;
END_REGION

REGION Network 22: DISK SPEED LINE 2 LIMITS CALCULATION WARNING
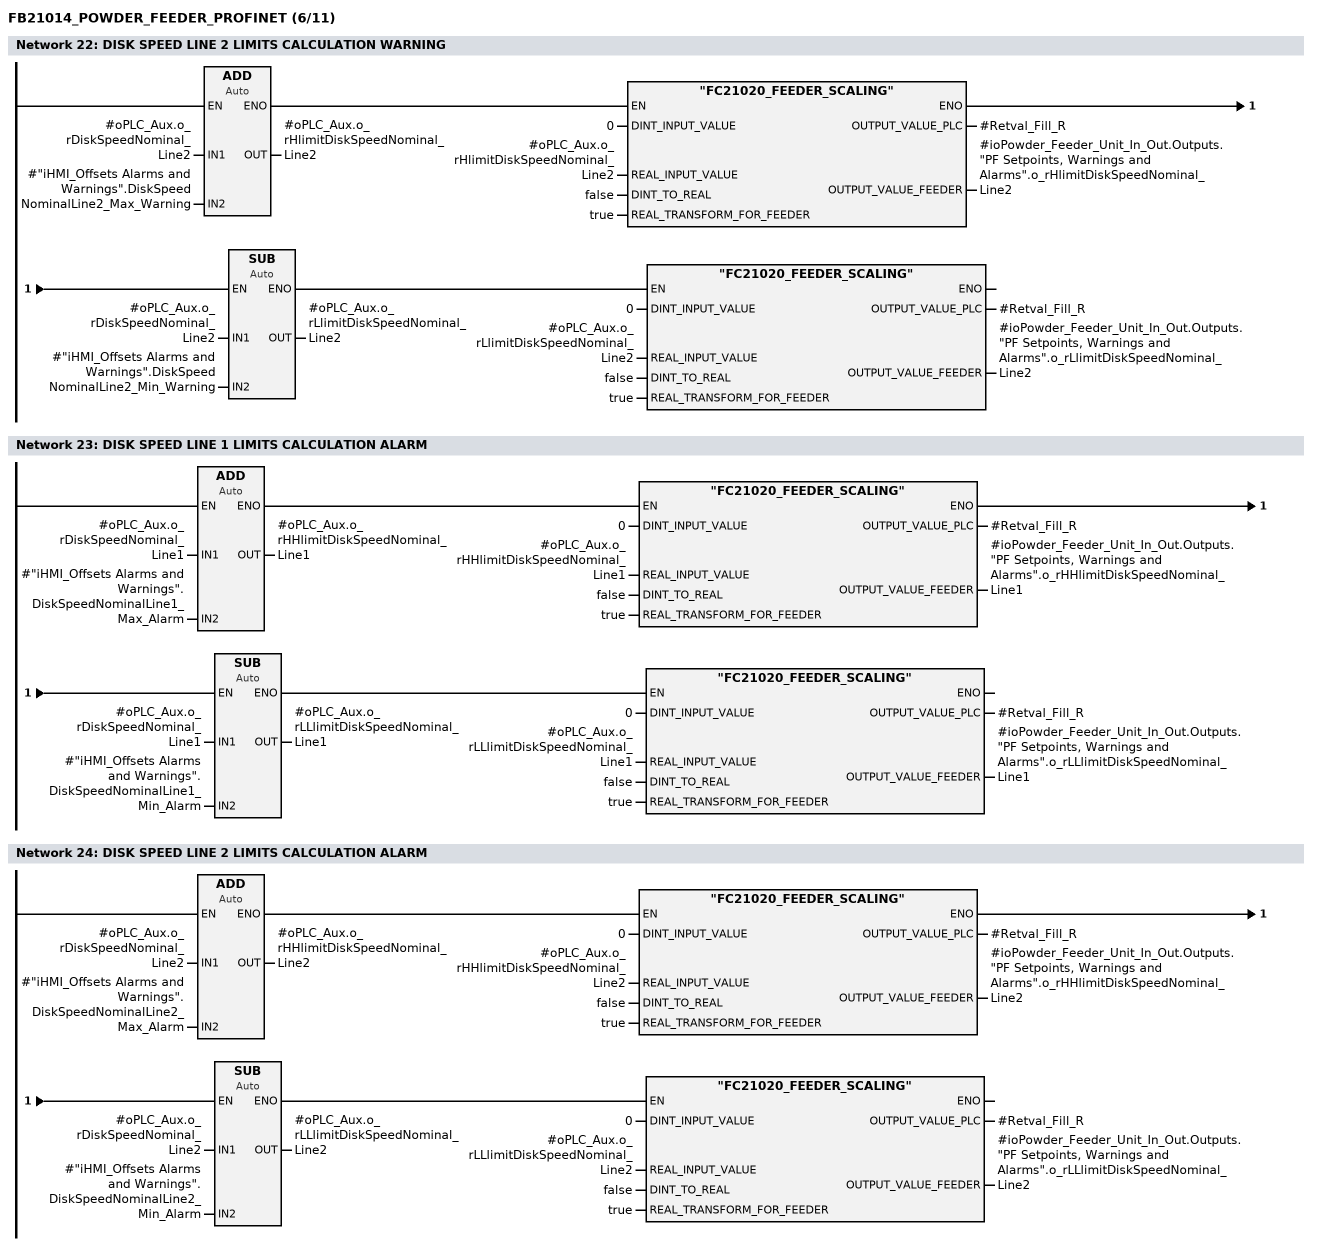
   RUNG wire#powerrail
      Add(in1 := #oPLC_Aux.o_rDiskSpeedNominal_Line2, in2 := #"iHMI_Offsets Alarms and Warnings".DiskSpeedNominalLine2_Max_Warning, out => #oPLC_Aux.o_rHlimitDiskSpeedNominal_Line2)
      "FC21020_FEEDER_SCALING"(DINT_INPUT_VALUE := 0, REAL_INPUT_VALUE := #oPLC_Aux.o_rHlimitDiskSpeedNominal_Line2, DINT_TO_REAL := false, REAL_TRANSFORM_FOR_FEEDER := true, OUTPUT_VALUE_PLC => #Retval_Fill_R, OUTPUT_VALUE_FEEDER => #ioPowder_Feeder_Unit_In_Out.Outputs."PF Setpoints, Warnings and Alarms".o_rHlimitDiskSpeedNominal_Line2)
      Sub(in1 := #oPLC_Aux.o_rDiskSpeedNominal_Line2, in2 := #"iHMI_Offsets Alarms and Warnings".DiskSpeedNominalLine2_Min_Warning, out => #oPLC_Aux.o_rLlimitDiskSpeedNominal_Line2)
      "FC21020_FEEDER_SCALING"(DINT_INPUT_VALUE := 0, REAL_INPUT_VALUE := #oPLC_Aux.o_rLlimitDiskSpeedNominal_Line2, DINT_TO_REAL := false, REAL_TRANSFORM_FOR_FEEDER := true, OUTPUT_VALUE_PLC => #Retval_Fill_R, OUTPUT_VALUE_FEEDER => #ioPowder_Feeder_Unit_In_Out.Outputs."PF Setpoints, Warnings and Alarms".o_rLlimitDiskSpeedNominal_Line2)
   END_RUNG
   // the same network as SCL:
   #oPLC_Aux.o_rHlimitDiskSpeedNominal_Line2 := #oPLC_Aux.o_rDiskSpeedNominal_Line2 + #"iHMI_Offsets Alarms and Warnings".DiskSpeedNominalLine2_Max_Warning;
   "FC21020_FEEDER_SCALING"(DINT_INPUT_VALUE := 0,
                           REAL_INPUT_VALUE := #oPLC_Aux.o_rHlimitDiskSpeedNominal_Line2,
                           DINT_TO_REAL := false,
                           REAL_TRANSFORM_FOR_FEEDER := true,
                           OUTPUT_VALUE_PLC => #Retval_Fill_R,
                           OUTPUT_VALUE_FEEDER => #ioPowder_Feeder_Unit_In_Out.Outputs."PF Setpoints, Warnings and Alarms".o_rHlimitDiskSpeedNominal_Line2,
                           ENO => #_w1);
   IF #_w1 THEN
       #oPLC_Aux.o_rLlimitDiskSpeedNominal_Line2 := #oPLC_Aux.o_rDiskSpeedNominal_Line2 - #"iHMI_Offsets Alarms and Warnings".DiskSpeedNominalLine2_Min_Warning;
       "FC21020_FEEDER_SCALING"(DINT_INPUT_VALUE := 0,
                               REAL_INPUT_VALUE := #oPLC_Aux.o_rLlimitDiskSpeedNominal_Line2,
                               DINT_TO_REAL := false,
                               REAL_TRANSFORM_FOR_FEEDER := true,
                               OUTPUT_VALUE_PLC => #Retval_Fill_R,
                               OUTPUT_VALUE_FEEDER => #ioPowder_Feeder_Unit_In_Out.Outputs."PF Setpoints, Warnings and Alarms".o_rLlimitDiskSpeedNominal_Line2);
   END_IF;
END_REGION

REGION Network 23: DISK SPEED LINE 1 LIMITS CALCULATION ALARM
   RUNG wire#powerrail
      Add(in1 := #oPLC_Aux.o_rDiskSpeedNominal_Line1, in2 := #"iHMI_Offsets Alarms and Warnings".DiskSpeedNominalLine1_Max_Alarm, out => #oPLC_Aux.o_rHHlimitDiskSpeedNominal_Line1)
      "FC21020_FEEDER_SCALING"(DINT_INPUT_VALUE := 0, REAL_INPUT_VALUE := #oPLC_Aux.o_rHHlimitDiskSpeedNominal_Line1, DINT_TO_REAL := false, REAL_TRANSFORM_FOR_FEEDER := true, OUTPUT_VALUE_PLC => #Retval_Fill_R, OUTPUT_VALUE_FEEDER => #ioPowder_Feeder_Unit_In_Out.Outputs."PF Setpoints, Warnings and Alarms".o_rHHlimitDiskSpeedNominal_Line1)
      Sub(in1 := #oPLC_Aux.o_rDiskSpeedNominal_Line1, in2 := #"iHMI_Offsets Alarms and Warnings".DiskSpeedNominalLine1_Min_Alarm, out => #oPLC_Aux.o_rLLlimitDiskSpeedNominal_Line1)
      "FC21020_FEEDER_SCALING"(DINT_INPUT_VALUE := 0, REAL_INPUT_VALUE := #oPLC_Aux.o_rLLlimitDiskSpeedNominal_Line1, DINT_TO_REAL := false, REAL_TRANSFORM_FOR_FEEDER := true, OUTPUT_VALUE_PLC => #Retval_Fill_R, OUTPUT_VALUE_FEEDER => #ioPowder_Feeder_Unit_In_Out.Outputs."PF Setpoints, Warnings and Alarms".o_rLLlimitDiskSpeedNominal_Line1)
   END_RUNG
   // the same network as SCL:
   #oPLC_Aux.o_rHHlimitDiskSpeedNominal_Line1 := #oPLC_Aux.o_rDiskSpeedNominal_Line1 + #"iHMI_Offsets Alarms and Warnings".DiskSpeedNominalLine1_Max_Alarm;
   "FC21020_FEEDER_SCALING"(DINT_INPUT_VALUE := 0,
                           REAL_INPUT_VALUE := #oPLC_Aux.o_rHHlimitDiskSpeedNominal_Line1,
                           DINT_TO_REAL := false,
                           REAL_TRANSFORM_FOR_FEEDER := true,
                           OUTPUT_VALUE_PLC => #Retval_Fill_R,
                           OUTPUT_VALUE_FEEDER => #ioPowder_Feeder_Unit_In_Out.Outputs."PF Setpoints, Warnings and Alarms".o_rHHlimitDiskSpeedNominal_Line1,
                           ENO => #_w1);
   IF #_w1 THEN
       #oPLC_Aux.o_rLLlimitDiskSpeedNominal_Line1 := #oPLC_Aux.o_rDiskSpeedNominal_Line1 - #"iHMI_Offsets Alarms and Warnings".DiskSpeedNominalLine1_Min_Alarm;
       "FC21020_FEEDER_SCALING"(DINT_INPUT_VALUE := 0,
                               REAL_INPUT_VALUE := #oPLC_Aux.o_rLLlimitDiskSpeedNominal_Line1,
                               DINT_TO_REAL := false,
                               REAL_TRANSFORM_FOR_FEEDER := true,
                               OUTPUT_VALUE_PLC => #Retval_Fill_R,
                               OUTPUT_VALUE_FEEDER => #ioPowder_Feeder_Unit_In_Out.Outputs."PF Setpoints, Warnings and Alarms".o_rLLlimitDiskSpeedNominal_Line1);
   END_IF;
END_REGION

REGION Network 24: DISK SPEED LINE 2 LIMITS CALCULATION ALARM
   RUNG wire#powerrail
      Add(in1 := #oPLC_Aux.o_rDiskSpeedNominal_Line2, in2 := #"iHMI_Offsets Alarms and Warnings".DiskSpeedNominalLine2_Max_Alarm, out => #oPLC_Aux.o_rHHlimitDiskSpeedNominal_Line2)
      "FC21020_FEEDER_SCALING"(DINT_INPUT_VALUE := 0, REAL_INPUT_VALUE := #oPLC_Aux.o_rHHlimitDiskSpeedNominal_Line2, DINT_TO_REAL := false, REAL_TRANSFORM_FOR_FEEDER := true, OUTPUT_VALUE_PLC => #Retval_Fill_R, OUTPUT_VALUE_FEEDER => #ioPowder_Feeder_Unit_In_Out.Outputs."PF Setpoints, Warnings and Alarms".o_rHHlimitDiskSpeedNominal_Line2)
      Sub(in1 := #oPLC_Aux.o_rDiskSpeedNominal_Line2, in2 := #"iHMI_Offsets Alarms and Warnings".DiskSpeedNominalLine2_Min_Alarm, out => #oPLC_Aux.o_rLLlimitDiskSpeedNominal_Line2)
      "FC21020_FEEDER_SCALING"(DINT_INPUT_VALUE := 0, REAL_INPUT_VALUE := #oPLC_Aux.o_rLLlimitDiskSpeedNominal_Line2, DINT_TO_REAL := false, REAL_TRANSFORM_FOR_FEEDER := true, OUTPUT_VALUE_PLC => #Retval_Fill_R, OUTPUT_VALUE_FEEDER => #ioPowder_Feeder_Unit_In_Out.Outputs."PF Setpoints, Warnings and Alarms".o_rLLlimitDiskSpeedNominal_Line2)
   END_RUNG
   // the same network as SCL:
   #oPLC_Aux.o_rHHlimitDiskSpeedNominal_Line2 := #oPLC_Aux.o_rDiskSpeedNominal_Line2 + #"iHMI_Offsets Alarms and Warnings".DiskSpeedNominalLine2_Max_Alarm;
   "FC21020_FEEDER_SCALING"(DINT_INPUT_VALUE := 0,
                           REAL_INPUT_VALUE := #oPLC_Aux.o_rHHlimitDiskSpeedNominal_Line2,
                           DINT_TO_REAL := false,
                           REAL_TRANSFORM_FOR_FEEDER := true,
                           OUTPUT_VALUE_PLC => #Retval_Fill_R,
                           OUTPUT_VALUE_FEEDER => #ioPowder_Feeder_Unit_In_Out.Outputs."PF Setpoints, Warnings and Alarms".o_rHHlimitDiskSpeedNominal_Line2,
                           ENO => #_w1);
   IF #_w1 THEN
       #oPLC_Aux.o_rLLlimitDiskSpeedNominal_Line2 := #oPLC_Aux.o_rDiskSpeedNominal_Line2 - #"iHMI_Offsets Alarms and Warnings".DiskSpeedNominalLine2_Min_Alarm;
       "FC21020_FEEDER_SCALING"(DINT_INPUT_VALUE := 0,
                               REAL_INPUT_VALUE := #oPLC_Aux.o_rLLlimitDiskSpeedNominal_Line2,
                               DINT_TO_REAL := false,
                               REAL_TRANSFORM_FOR_FEEDER := true,
                               OUTPUT_VALUE_PLC => #Retval_Fill_R,
                               OUTPUT_VALUE_FEEDER => #ioPowder_Feeder_Unit_In_Out.Outputs."PF Setpoints, Warnings and Alarms".o_rLLlimitDiskSpeedNominal_Line2);
   END_IF;
END_REGION

REGION Network 25: STIRRER SPEED LINE 1 LIMITS CALCULATION WARNING
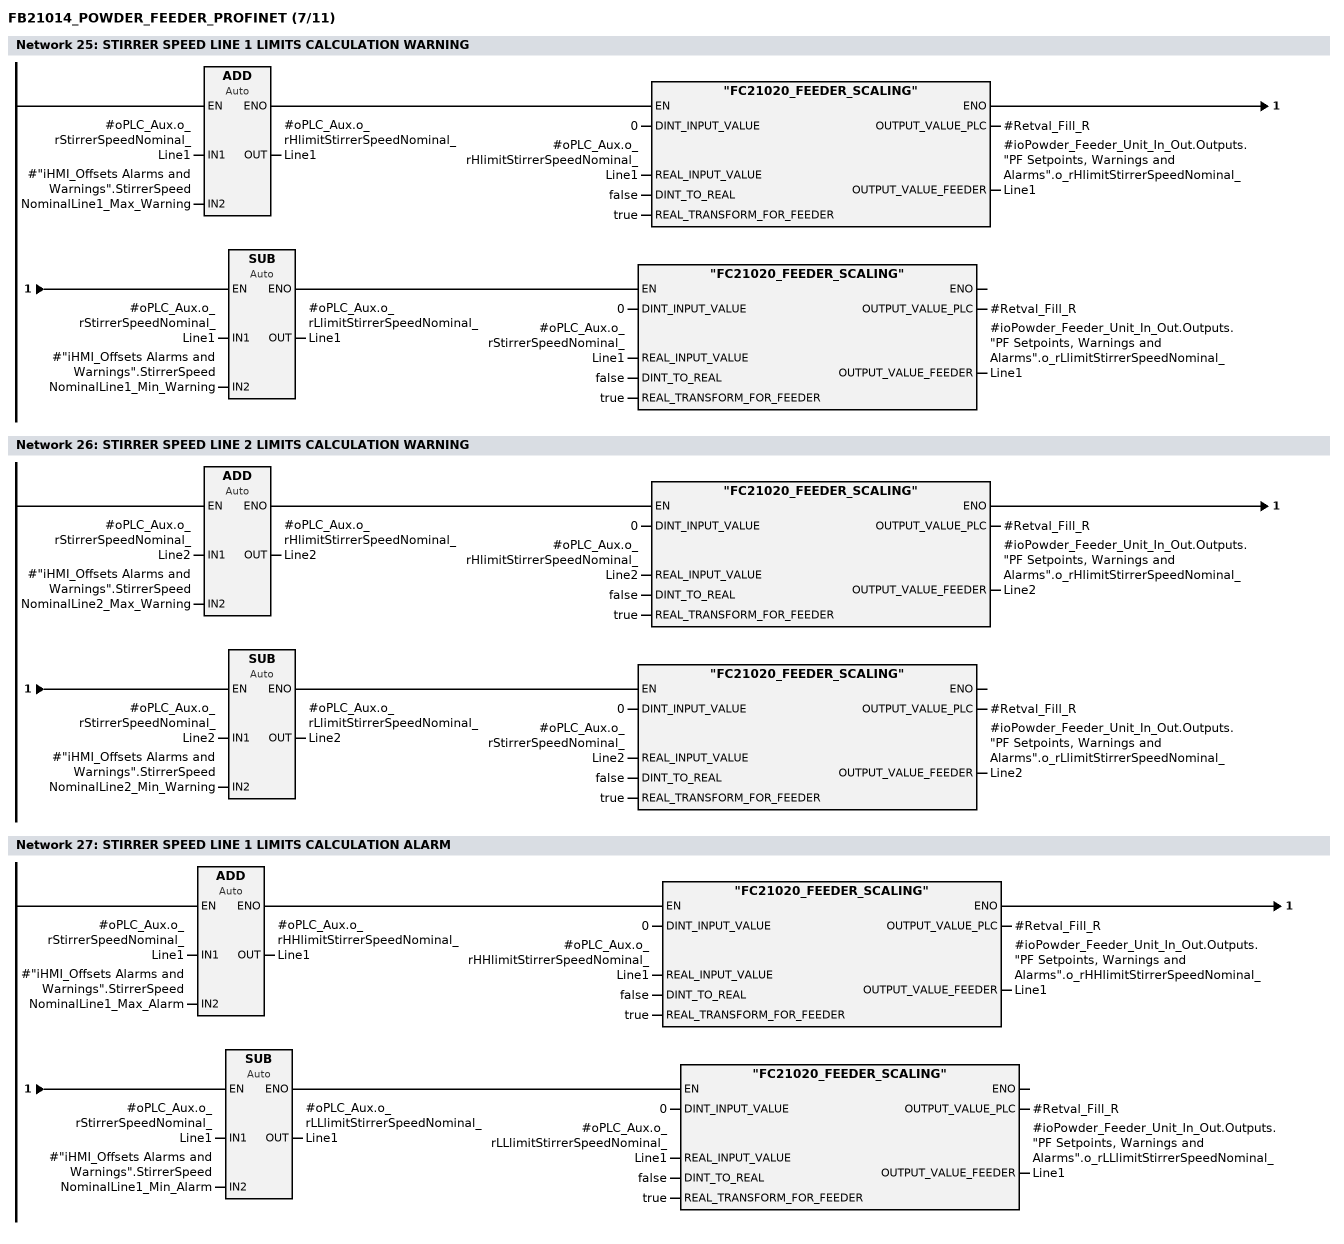
   RUNG wire#powerrail
      Add(in1 := #oPLC_Aux.o_rStirrerSpeedNominal_Line1, in2 := #"iHMI_Offsets Alarms and Warnings".StirrerSpeedNominalLine1_Max_Warning, out => #oPLC_Aux.o_rHlimitStirrerSpeedNominal_Line1)
      "FC21020_FEEDER_SCALING"(DINT_INPUT_VALUE := 0, REAL_INPUT_VALUE := #oPLC_Aux.o_rHlimitStirrerSpeedNominal_Line1, DINT_TO_REAL := false, REAL_TRANSFORM_FOR_FEEDER := true, OUTPUT_VALUE_PLC => #Retval_Fill_R, OUTPUT_VALUE_FEEDER => #ioPowder_Feeder_Unit_In_Out.Outputs."PF Setpoints, Warnings and Alarms".o_rHlimitStirrerSpeedNominal_Line1)
      Sub(in1 := #oPLC_Aux.o_rStirrerSpeedNominal_Line1, in2 := #"iHMI_Offsets Alarms and Warnings".StirrerSpeedNominalLine1_Min_Warning, out => #oPLC_Aux.o_rLlimitStirrerSpeedNominal_Line1)
      "FC21020_FEEDER_SCALING"(DINT_INPUT_VALUE := 0, REAL_INPUT_VALUE := #oPLC_Aux.o_rStirrerSpeedNominal_Line1, DINT_TO_REAL := false, REAL_TRANSFORM_FOR_FEEDER := true, OUTPUT_VALUE_PLC => #Retval_Fill_R, OUTPUT_VALUE_FEEDER => #ioPowder_Feeder_Unit_In_Out.Outputs."PF Setpoints, Warnings and Alarms".o_rLlimitStirrerSpeedNominal_Line1)
   END_RUNG
   // the same network as SCL:
   #oPLC_Aux.o_rHlimitStirrerSpeedNominal_Line1 := #oPLC_Aux.o_rStirrerSpeedNominal_Line1 + #"iHMI_Offsets Alarms and Warnings".StirrerSpeedNominalLine1_Max_Warning;
   "FC21020_FEEDER_SCALING"(DINT_INPUT_VALUE := 0,
                           REAL_INPUT_VALUE := #oPLC_Aux.o_rHlimitStirrerSpeedNominal_Line1,
                           DINT_TO_REAL := false,
                           REAL_TRANSFORM_FOR_FEEDER := true,
                           OUTPUT_VALUE_PLC => #Retval_Fill_R,
                           OUTPUT_VALUE_FEEDER => #ioPowder_Feeder_Unit_In_Out.Outputs."PF Setpoints, Warnings and Alarms".o_rHlimitStirrerSpeedNominal_Line1,
                           ENO => #_w1);
   IF #_w1 THEN
       #oPLC_Aux.o_rLlimitStirrerSpeedNominal_Line1 := #oPLC_Aux.o_rStirrerSpeedNominal_Line1 - #"iHMI_Offsets Alarms and Warnings".StirrerSpeedNominalLine1_Min_Warning;
       "FC21020_FEEDER_SCALING"(DINT_INPUT_VALUE := 0,
                               REAL_INPUT_VALUE := #oPLC_Aux.o_rStirrerSpeedNominal_Line1,
                               DINT_TO_REAL := false,
                               REAL_TRANSFORM_FOR_FEEDER := true,
                               OUTPUT_VALUE_PLC => #Retval_Fill_R,
                               OUTPUT_VALUE_FEEDER => #ioPowder_Feeder_Unit_In_Out.Outputs."PF Setpoints, Warnings and Alarms".o_rLlimitStirrerSpeedNominal_Line1);
   END_IF;
END_REGION

REGION Network 26: STIRRER SPEED LINE 2 LIMITS CALCULATION WARNING
   RUNG wire#powerrail
      Add(in1 := #oPLC_Aux.o_rStirrerSpeedNominal_Line2, in2 := #"iHMI_Offsets Alarms and Warnings".StirrerSpeedNominalLine2_Max_Warning, out => #oPLC_Aux.o_rHlimitStirrerSpeedNominal_Line2)
      "FC21020_FEEDER_SCALING"(DINT_INPUT_VALUE := 0, REAL_INPUT_VALUE := #oPLC_Aux.o_rHlimitStirrerSpeedNominal_Line2, DINT_TO_REAL := false, REAL_TRANSFORM_FOR_FEEDER := true, OUTPUT_VALUE_PLC => #Retval_Fill_R, OUTPUT_VALUE_FEEDER => #ioPowder_Feeder_Unit_In_Out.Outputs."PF Setpoints, Warnings and Alarms".o_rHlimitStirrerSpeedNominal_Line2)
      Sub(in1 := #oPLC_Aux.o_rStirrerSpeedNominal_Line2, in2 := #"iHMI_Offsets Alarms and Warnings".StirrerSpeedNominalLine2_Min_Warning, out => #oPLC_Aux.o_rLlimitStirrerSpeedNominal_Line2)
      "FC21020_FEEDER_SCALING"(DINT_INPUT_VALUE := 0, REAL_INPUT_VALUE := #oPLC_Aux.o_rStirrerSpeedNominal_Line2, DINT_TO_REAL := false, REAL_TRANSFORM_FOR_FEEDER := true, OUTPUT_VALUE_PLC => #Retval_Fill_R, OUTPUT_VALUE_FEEDER => #ioPowder_Feeder_Unit_In_Out.Outputs."PF Setpoints, Warnings and Alarms".o_rLlimitStirrerSpeedNominal_Line2)
   END_RUNG
   // the same network as SCL:
   #oPLC_Aux.o_rHlimitStirrerSpeedNominal_Line2 := #oPLC_Aux.o_rStirrerSpeedNominal_Line2 + #"iHMI_Offsets Alarms and Warnings".StirrerSpeedNominalLine2_Max_Warning;
   "FC21020_FEEDER_SCALING"(DINT_INPUT_VALUE := 0,
                           REAL_INPUT_VALUE := #oPLC_Aux.o_rHlimitStirrerSpeedNominal_Line2,
                           DINT_TO_REAL := false,
                           REAL_TRANSFORM_FOR_FEEDER := true,
                           OUTPUT_VALUE_PLC => #Retval_Fill_R,
                           OUTPUT_VALUE_FEEDER => #ioPowder_Feeder_Unit_In_Out.Outputs."PF Setpoints, Warnings and Alarms".o_rHlimitStirrerSpeedNominal_Line2,
                           ENO => #_w1);
   IF #_w1 THEN
       #oPLC_Aux.o_rLlimitStirrerSpeedNominal_Line2 := #oPLC_Aux.o_rStirrerSpeedNominal_Line2 - #"iHMI_Offsets Alarms and Warnings".StirrerSpeedNominalLine2_Min_Warning;
       "FC21020_FEEDER_SCALING"(DINT_INPUT_VALUE := 0,
                               REAL_INPUT_VALUE := #oPLC_Aux.o_rStirrerSpeedNominal_Line2,
                               DINT_TO_REAL := false,
                               REAL_TRANSFORM_FOR_FEEDER := true,
                               OUTPUT_VALUE_PLC => #Retval_Fill_R,
                               OUTPUT_VALUE_FEEDER => #ioPowder_Feeder_Unit_In_Out.Outputs."PF Setpoints, Warnings and Alarms".o_rLlimitStirrerSpeedNominal_Line2);
   END_IF;
END_REGION

REGION Network 27: STIRRER SPEED LINE 1 LIMITS CALCULATION ALARM
   RUNG wire#powerrail
      Add(in1 := #oPLC_Aux.o_rStirrerSpeedNominal_Line1, in2 := #"iHMI_Offsets Alarms and Warnings".StirrerSpeedNominalLine1_Max_Alarm, out => #oPLC_Aux.o_rHHlimitStirrerSpeedNominal_Line1)
      "FC21020_FEEDER_SCALING"(DINT_INPUT_VALUE := 0, REAL_INPUT_VALUE := #oPLC_Aux.o_rHHlimitStirrerSpeedNominal_Line1, DINT_TO_REAL := false, REAL_TRANSFORM_FOR_FEEDER := true, OUTPUT_VALUE_PLC => #Retval_Fill_R, OUTPUT_VALUE_FEEDER => #ioPowder_Feeder_Unit_In_Out.Outputs."PF Setpoints, Warnings and Alarms".o_rHHlimitStirrerSpeedNominal_Line1)
      Sub(in1 := #oPLC_Aux.o_rStirrerSpeedNominal_Line1, in2 := #"iHMI_Offsets Alarms and Warnings".StirrerSpeedNominalLine1_Min_Alarm, out => #oPLC_Aux.o_rLLlimitStirrerSpeedNominal_Line1)
      "FC21020_FEEDER_SCALING"(DINT_INPUT_VALUE := 0, REAL_INPUT_VALUE := #oPLC_Aux.o_rLLlimitStirrerSpeedNominal_Line1, DINT_TO_REAL := false, REAL_TRANSFORM_FOR_FEEDER := true, OUTPUT_VALUE_PLC => #Retval_Fill_R, OUTPUT_VALUE_FEEDER => #ioPowder_Feeder_Unit_In_Out.Outputs."PF Setpoints, Warnings and Alarms".o_rLLlimitStirrerSpeedNominal_Line1)
   END_RUNG
   // the same network as SCL:
   #oPLC_Aux.o_rHHlimitStirrerSpeedNominal_Line1 := #oPLC_Aux.o_rStirrerSpeedNominal_Line1 + #"iHMI_Offsets Alarms and Warnings".StirrerSpeedNominalLine1_Max_Alarm;
   "FC21020_FEEDER_SCALING"(DINT_INPUT_VALUE := 0,
                           REAL_INPUT_VALUE := #oPLC_Aux.o_rHHlimitStirrerSpeedNominal_Line1,
                           DINT_TO_REAL := false,
                           REAL_TRANSFORM_FOR_FEEDER := true,
                           OUTPUT_VALUE_PLC => #Retval_Fill_R,
                           OUTPUT_VALUE_FEEDER => #ioPowder_Feeder_Unit_In_Out.Outputs."PF Setpoints, Warnings and Alarms".o_rHHlimitStirrerSpeedNominal_Line1,
                           ENO => #_w1);
   IF #_w1 THEN
       #oPLC_Aux.o_rLLlimitStirrerSpeedNominal_Line1 := #oPLC_Aux.o_rStirrerSpeedNominal_Line1 - #"iHMI_Offsets Alarms and Warnings".StirrerSpeedNominalLine1_Min_Alarm;
       "FC21020_FEEDER_SCALING"(DINT_INPUT_VALUE := 0,
                               REAL_INPUT_VALUE := #oPLC_Aux.o_rLLlimitStirrerSpeedNominal_Line1,
                               DINT_TO_REAL := false,
                               REAL_TRANSFORM_FOR_FEEDER := true,
                               OUTPUT_VALUE_PLC => #Retval_Fill_R,
                               OUTPUT_VALUE_FEEDER => #ioPowder_Feeder_Unit_In_Out.Outputs."PF Setpoints, Warnings and Alarms".o_rLLlimitStirrerSpeedNominal_Line1);
   END_IF;
END_REGION

REGION Network 28: STIRRER SPEED LINE 2 LIMITS CALCULATION ALARM
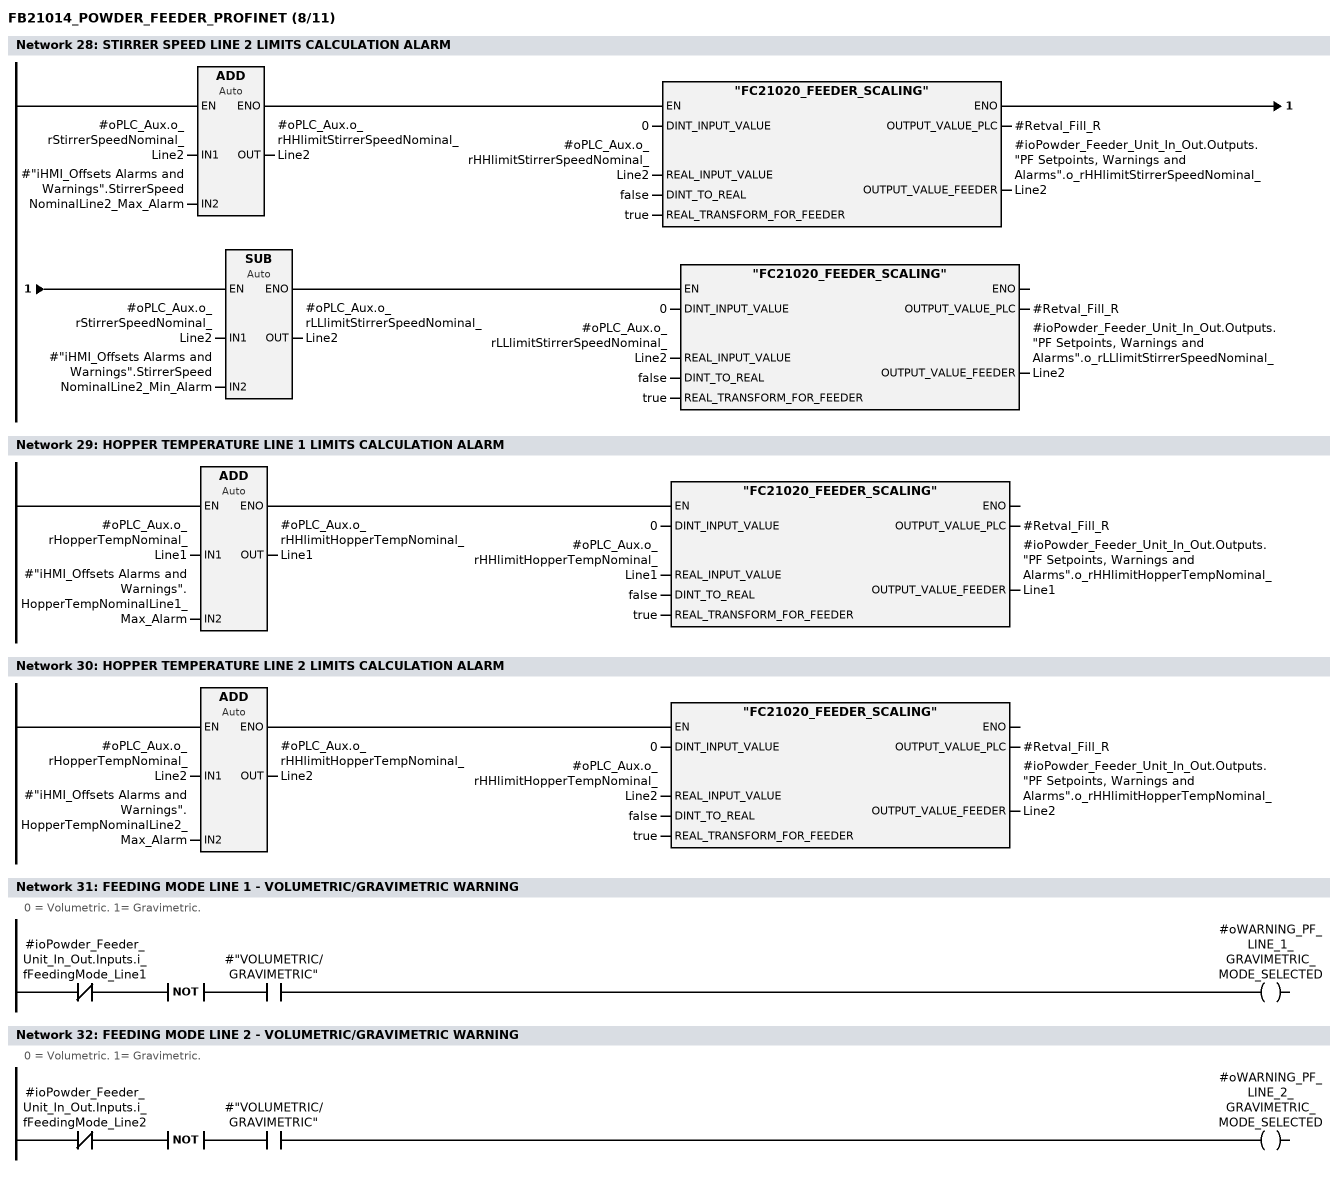
   RUNG wire#powerrail
      Add(in1 := #oPLC_Aux.o_rStirrerSpeedNominal_Line2, in2 := #"iHMI_Offsets Alarms and Warnings".StirrerSpeedNominalLine2_Max_Alarm, out => #oPLC_Aux.o_rHHlimitStirrerSpeedNominal_Line2)
      "FC21020_FEEDER_SCALING"(DINT_INPUT_VALUE := 0, REAL_INPUT_VALUE := #oPLC_Aux.o_rHHlimitStirrerSpeedNominal_Line2, DINT_TO_REAL := false, REAL_TRANSFORM_FOR_FEEDER := true, OUTPUT_VALUE_PLC => #Retval_Fill_R, OUTPUT_VALUE_FEEDER => #ioPowder_Feeder_Unit_In_Out.Outputs."PF Setpoints, Warnings and Alarms".o_rHHlimitStirrerSpeedNominal_Line2)
      Sub(in1 := #oPLC_Aux.o_rStirrerSpeedNominal_Line2, in2 := #"iHMI_Offsets Alarms and Warnings".StirrerSpeedNominalLine2_Min_Alarm, out => #oPLC_Aux.o_rLLlimitStirrerSpeedNominal_Line2)
      "FC21020_FEEDER_SCALING"(DINT_INPUT_VALUE := 0, REAL_INPUT_VALUE := #oPLC_Aux.o_rLLlimitStirrerSpeedNominal_Line2, DINT_TO_REAL := false, REAL_TRANSFORM_FOR_FEEDER := true, OUTPUT_VALUE_PLC => #Retval_Fill_R, OUTPUT_VALUE_FEEDER => #ioPowder_Feeder_Unit_In_Out.Outputs."PF Setpoints, Warnings and Alarms".o_rLLlimitStirrerSpeedNominal_Line2)
   END_RUNG
   // the same network as SCL:
   #oPLC_Aux.o_rHHlimitStirrerSpeedNominal_Line2 := #oPLC_Aux.o_rStirrerSpeedNominal_Line2 + #"iHMI_Offsets Alarms and Warnings".StirrerSpeedNominalLine2_Max_Alarm;
   "FC21020_FEEDER_SCALING"(DINT_INPUT_VALUE := 0,
                           REAL_INPUT_VALUE := #oPLC_Aux.o_rHHlimitStirrerSpeedNominal_Line2,
                           DINT_TO_REAL := false,
                           REAL_TRANSFORM_FOR_FEEDER := true,
                           OUTPUT_VALUE_PLC => #Retval_Fill_R,
                           OUTPUT_VALUE_FEEDER => #ioPowder_Feeder_Unit_In_Out.Outputs."PF Setpoints, Warnings and Alarms".o_rHHlimitStirrerSpeedNominal_Line2,
                           ENO => #_w1);
   IF #_w1 THEN
       #oPLC_Aux.o_rLLlimitStirrerSpeedNominal_Line2 := #oPLC_Aux.o_rStirrerSpeedNominal_Line2 - #"iHMI_Offsets Alarms and Warnings".StirrerSpeedNominalLine2_Min_Alarm;
       "FC21020_FEEDER_SCALING"(DINT_INPUT_VALUE := 0,
                               REAL_INPUT_VALUE := #oPLC_Aux.o_rLLlimitStirrerSpeedNominal_Line2,
                               DINT_TO_REAL := false,
                               REAL_TRANSFORM_FOR_FEEDER := true,
                               OUTPUT_VALUE_PLC => #Retval_Fill_R,
                               OUTPUT_VALUE_FEEDER => #ioPowder_Feeder_Unit_In_Out.Outputs."PF Setpoints, Warnings and Alarms".o_rLLlimitStirrerSpeedNominal_Line2);
   END_IF;
END_REGION

REGION Network 29: HOPPER TEMPERATURE LINE 1 LIMITS CALCULATION ALARM
   RUNG wire#powerrail
      Add(in1 := #oPLC_Aux.o_rHopperTempNominal_Line1, in2 := #"iHMI_Offsets Alarms and Warnings".HopperTempNominalLine1_Max_Alarm, out => #oPLC_Aux.o_rHHlimitHopperTempNominal_Line1)
      "FC21020_FEEDER_SCALING"(DINT_INPUT_VALUE := 0, REAL_INPUT_VALUE := #oPLC_Aux.o_rHHlimitHopperTempNominal_Line1, DINT_TO_REAL := false, REAL_TRANSFORM_FOR_FEEDER := true, OUTPUT_VALUE_PLC => #Retval_Fill_R, OUTPUT_VALUE_FEEDER => #ioPowder_Feeder_Unit_In_Out.Outputs."PF Setpoints, Warnings and Alarms".o_rHHlimitHopperTempNominal_Line1)
   END_RUNG
   // the same network as SCL:
   #oPLC_Aux.o_rHHlimitHopperTempNominal_Line1 := #oPLC_Aux.o_rHopperTempNominal_Line1 + #"iHMI_Offsets Alarms and Warnings".HopperTempNominalLine1_Max_Alarm;
   "FC21020_FEEDER_SCALING"(DINT_INPUT_VALUE := 0,
                           REAL_INPUT_VALUE := #oPLC_Aux.o_rHHlimitHopperTempNominal_Line1,
                           DINT_TO_REAL := false,
                           REAL_TRANSFORM_FOR_FEEDER := true,
                           OUTPUT_VALUE_PLC => #Retval_Fill_R,
                           OUTPUT_VALUE_FEEDER => #ioPowder_Feeder_Unit_In_Out.Outputs."PF Setpoints, Warnings and Alarms".o_rHHlimitHopperTempNominal_Line1);
END_REGION

REGION Network 30: HOPPER TEMPERATURE LINE 2 LIMITS CALCULATION ALARM
   RUNG wire#powerrail
      Add(in1 := #oPLC_Aux.o_rHopperTempNominal_Line2, in2 := #"iHMI_Offsets Alarms and Warnings".HopperTempNominalLine2_Max_Alarm, out => #oPLC_Aux.o_rHHlimitHopperTempNominal_Line2)
      "FC21020_FEEDER_SCALING"(DINT_INPUT_VALUE := 0, REAL_INPUT_VALUE := #oPLC_Aux.o_rHHlimitHopperTempNominal_Line2, DINT_TO_REAL := false, REAL_TRANSFORM_FOR_FEEDER := true, OUTPUT_VALUE_PLC => #Retval_Fill_R, OUTPUT_VALUE_FEEDER => #ioPowder_Feeder_Unit_In_Out.Outputs."PF Setpoints, Warnings and Alarms".o_rHHlimitHopperTempNominal_Line2)
   END_RUNG
   // the same network as SCL:
   #oPLC_Aux.o_rHHlimitHopperTempNominal_Line2 := #oPLC_Aux.o_rHopperTempNominal_Line2 + #"iHMI_Offsets Alarms and Warnings".HopperTempNominalLine2_Max_Alarm;
   "FC21020_FEEDER_SCALING"(DINT_INPUT_VALUE := 0,
                           REAL_INPUT_VALUE := #oPLC_Aux.o_rHHlimitHopperTempNominal_Line2,
                           DINT_TO_REAL := false,
                           REAL_TRANSFORM_FOR_FEEDER := true,
                           OUTPUT_VALUE_PLC => #Retval_Fill_R,
                           OUTPUT_VALUE_FEEDER => #ioPowder_Feeder_Unit_In_Out.Outputs."PF Setpoints, Warnings and Alarms".o_rHHlimitHopperTempNominal_Line2);
END_REGION

REGION Network 31: FEEDING MODE LINE 1 - VOLUMETRIC/GRAVIMETRIC WARNING
   // 0 = Volumetric. 1= Gravimetric.
   RUNG wire#powerrail
      I_Contact( #ioPowder_Feeder_Unit_In_Out.Inputs.i_fFeedingMode_Line1 )
      Not()
      Contact( #"VOLUMETRIC/GRAVIMETRIC" )
      Coil( #oWARNING_PF_LINE_1_GRAVIMETRIC_MODE_SELECTED )
   END_RUNG
   // the same network as SCL:
   #oWARNING_PF_LINE_1_GRAVIMETRIC_MODE_SELECTED := NOT (NOT #ioPowder_Feeder_Unit_In_Out.Inputs.i_fFeedingMode_Line1) AND #"VOLUMETRIC/GRAVIMETRIC";
END_REGION

REGION Network 32: FEEDING MODE LINE 2 - VOLUMETRIC/GRAVIMETRIC WARNING
   // 0 = Volumetric. 1= Gravimetric.
   RUNG wire#powerrail
      I_Contact( #ioPowder_Feeder_Unit_In_Out.Inputs.i_fFeedingMode_Line2 )
      Not()
      Contact( #"VOLUMETRIC/GRAVIMETRIC" )
      Coil( #oWARNING_PF_LINE_2_GRAVIMETRIC_MODE_SELECTED )
   END_RUNG
   // the same network as SCL:
   #oWARNING_PF_LINE_2_GRAVIMETRIC_MODE_SELECTED := NOT (NOT #ioPowder_Feeder_Unit_In_Out.Inputs.i_fFeedingMode_Line2) AND #"VOLUMETRIC/GRAVIMETRIC";
END_REGION

REGION Network 33: WARNING
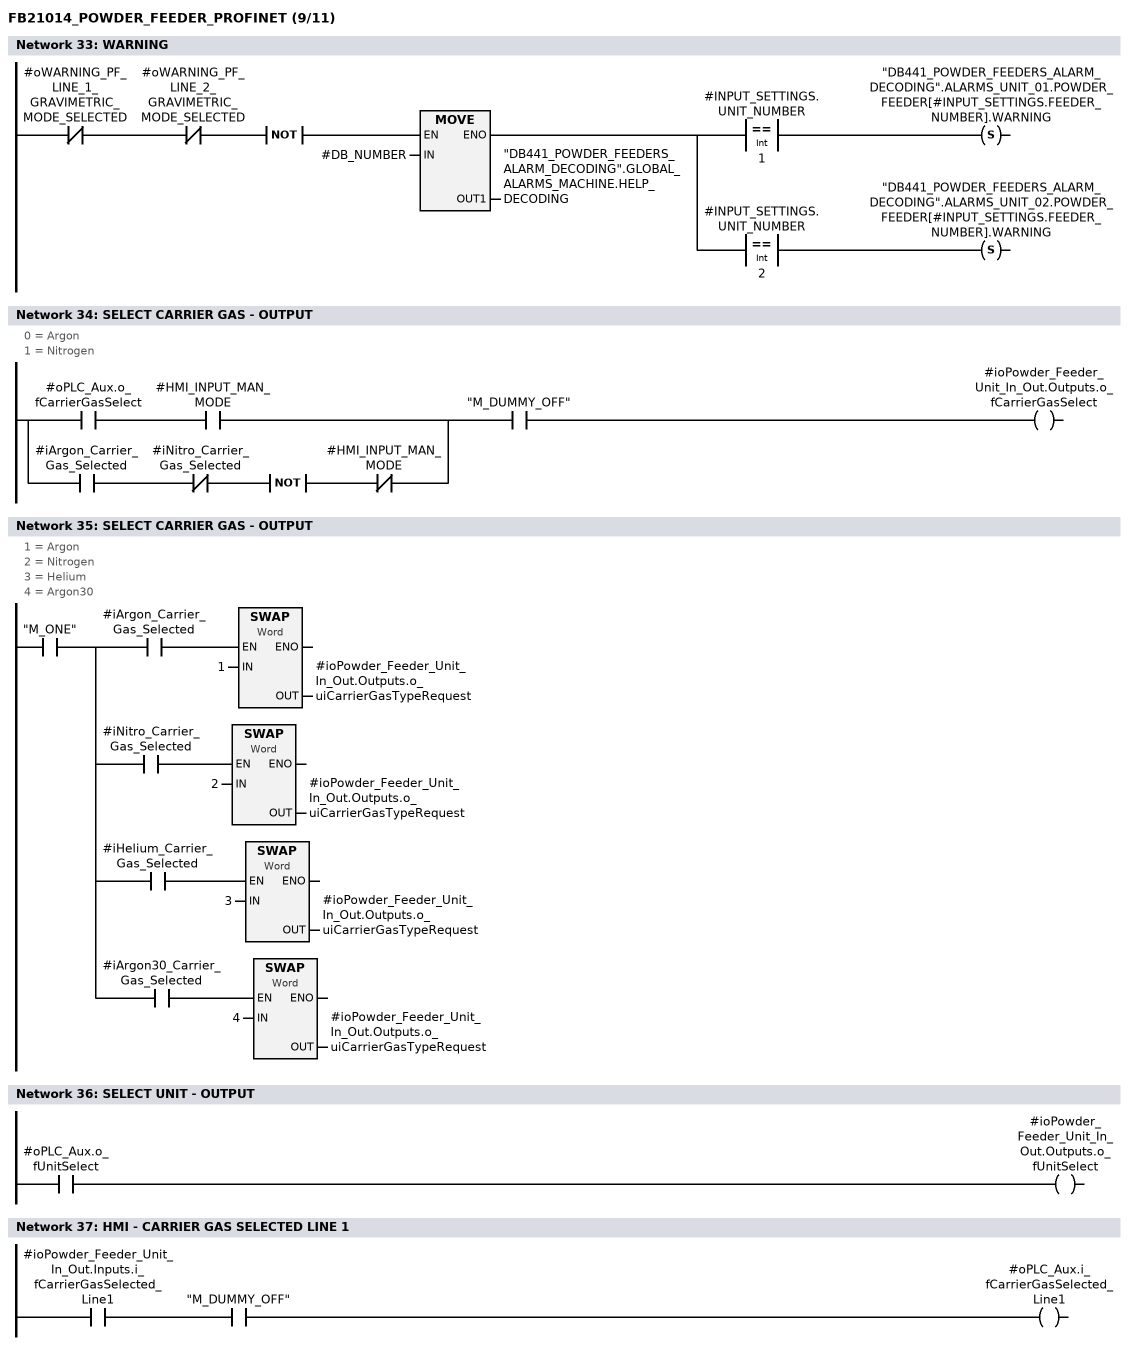
   RUNG wire#powerrail
      I_Contact( #oWARNING_PF_LINE_1_GRAVIMETRIC_MODE_SELECTED )
      I_Contact( #oWARNING_PF_LINE_2_GRAVIMETRIC_MODE_SELECTED )
      Not()
      Move(in := #DB_NUMBER, out1 => "DB441_POWDER_FEEDERS_ALARM_DECODING".GLOBAL_ALARMS_MACHINE.HELP_DECODING)
      wire#w1
      { S7_Templates := "SrcType := Int" } EQ_Contact(in1 := #INPUT_SETTINGS.UNIT_NUMBER, in2 := 1)
      S_Coil( "DB441_POWDER_FEEDERS_ALARM_DECODING".ALARMS_UNIT_01.POWDER_FEEDER[#INPUT_SETTINGS.FEEDER_NUMBER].WARNING )
   END_RUNG
   RUNG wire#w1
      { S7_Templates := "SrcType := Int" } EQ_Contact(in1 := #INPUT_SETTINGS.UNIT_NUMBER, in2 := 2)
      S_Coil( "DB441_POWDER_FEEDERS_ALARM_DECODING".ALARMS_UNIT_02.POWDER_FEEDER[#INPUT_SETTINGS.FEEDER_NUMBER].WARNING )
   END_RUNG
   // the same network as SCL:
   #_w1 := NOT (NOT #oWARNING_PF_LINE_1_GRAVIMETRIC_MODE_SELECTED AND NOT #oWARNING_PF_LINE_2_GRAVIMETRIC_MODE_SELECTED);
   IF #_w1 THEN
       "DB441_POWDER_FEEDERS_ALARM_DECODING".GLOBAL_ALARMS_MACHINE.HELP_DECODING := #DB_NUMBER;
   END_IF;
   IF #_w1 AND (#INPUT_SETTINGS.UNIT_NUMBER = 1) THEN
       "DB441_POWDER_FEEDERS_ALARM_DECODING".ALARMS_UNIT_01.POWDER_FEEDER[#INPUT_SETTINGS.FEEDER_NUMBER].WARNING := TRUE;
   END_IF;
   IF #_w1 AND (#INPUT_SETTINGS.UNIT_NUMBER = 2) THEN
       "DB441_POWDER_FEEDERS_ALARM_DECODING".ALARMS_UNIT_02.POWDER_FEEDER[#INPUT_SETTINGS.FEEDER_NUMBER].WARNING := TRUE;
   END_IF;
END_REGION

REGION Network 34: SELECT CARRIER GAS - OUTPUT
   // 0 = Argon
   // 1 = Nitrogen
   RUNG wire#powerrail
      Contact( #oPLC_Aux.o_fCarrierGasSelect )
      Contact( #HMI_INPUT_MAN_MODE )
      wire#w1
      Contact( "M_DUMMY_OFF" )
      Coil( #ioPowder_Feeder_Unit_In_Out.Outputs.o_fCarrierGasSelect )
   END_RUNG
   RUNG wire#powerrail
      Contact( #iArgon_Carrier_Gas_Selected )
      I_Contact( #iNitro_Carrier_Gas_Selected )
      Not()
      I_Contact( #HMI_INPUT_MAN_MODE )
   END_RUNG wire#w1
   // the same network as SCL:
   #ioPowder_Feeder_Unit_In_Out.Outputs.o_fCarrierGasSelect := ((#oPLC_Aux.o_fCarrierGasSelect AND #HMI_INPUT_MAN_MODE) OR (NOT (#iArgon_Carrier_Gas_Selected AND NOT #iNitro_Carrier_Gas_Selected) AND NOT #HMI_INPUT_MAN_MODE)) AND "M_DUMMY_OFF";
END_REGION

REGION Network 35: SELECT CARRIER GAS - OUTPUT
   // 1 = Argon
   // 2 = Nitrogen
   // 3 = Helium
   // 4 = Argon30
   IF "M_ONE" AND #iArgon_Carrier_Gas_Selected THEN
       #ioPowder_Feeder_Unit_In_Out.Outputs.o_uiCarrierGasTypeRequest := SWAP(1);
   END_IF;
   IF "M_ONE" AND #iNitro_Carrier_Gas_Selected THEN
       #ioPowder_Feeder_Unit_In_Out.Outputs.o_uiCarrierGasTypeRequest := SWAP(2);
   END_IF;
   IF "M_ONE" AND #iHelium_Carrier_Gas_Selected THEN
       #ioPowder_Feeder_Unit_In_Out.Outputs.o_uiCarrierGasTypeRequest := SWAP(3);
   END_IF;
   IF "M_ONE" AND #iArgon30_Carrier_Gas_Selected THEN
       #ioPowder_Feeder_Unit_In_Out.Outputs.o_uiCarrierGasTypeRequest := SWAP(4);
   END_IF;
END_REGION

REGION Network 36: SELECT UNIT - OUTPUT
   RUNG wire#powerrail
      Contact( #oPLC_Aux.o_fUnitSelect )
      Coil( #ioPowder_Feeder_Unit_In_Out.Outputs.o_fUnitSelect )
   END_RUNG
   // the same network as SCL:
   #ioPowder_Feeder_Unit_In_Out.Outputs.o_fUnitSelect := #oPLC_Aux.o_fUnitSelect;
END_REGION

REGION Network 37: HMI - CARRIER GAS SELECTED LINE 1
   RUNG wire#powerrail
      Contact( #ioPowder_Feeder_Unit_In_Out.Inputs.i_fCarrierGasSelected_Line1 )
      Contact( "M_DUMMY_OFF" )
      Coil( #oPLC_Aux.i_fCarrierGasSelected_Line1 )
   END_RUNG
   // the same network as SCL:
   #oPLC_Aux.i_fCarrierGasSelected_Line1 := #ioPowder_Feeder_Unit_In_Out.Inputs.i_fCarrierGasSelected_Line1 AND "M_DUMMY_OFF";
END_REGION

REGION Network 38: HMI - CARRIER GAS SELECTED LINE 2
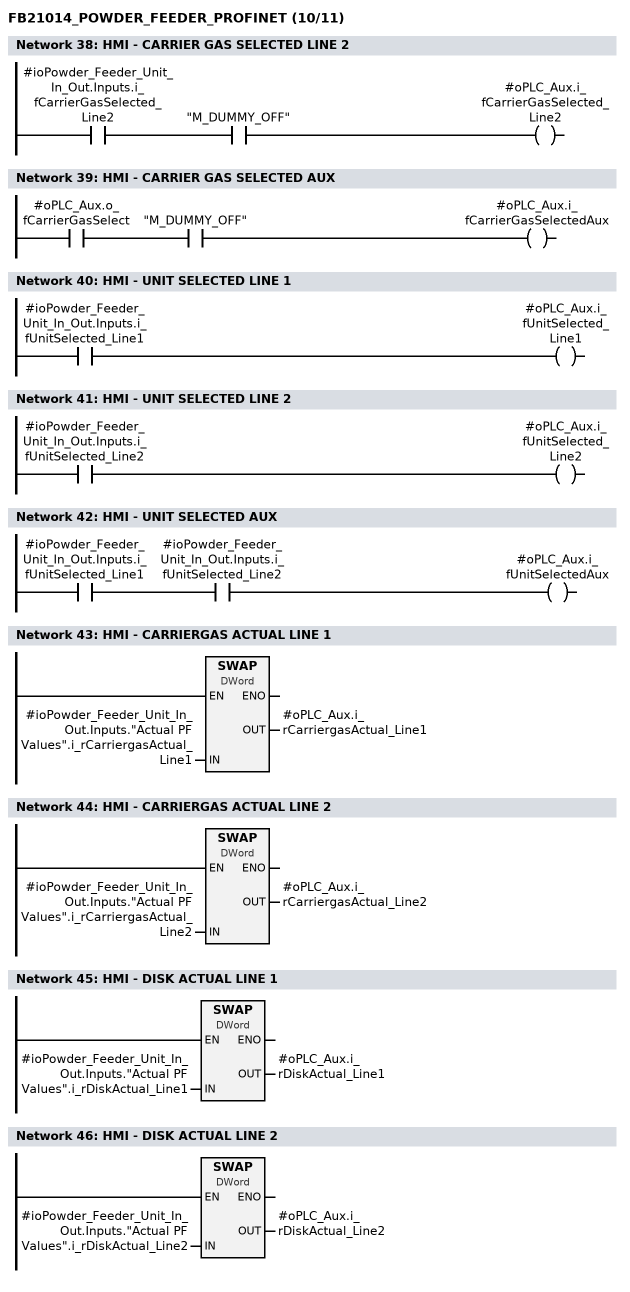
   RUNG wire#powerrail
      Contact( #ioPowder_Feeder_Unit_In_Out.Inputs.i_fCarrierGasSelected_Line2 )
      Contact( "M_DUMMY_OFF" )
      Coil( #oPLC_Aux.i_fCarrierGasSelected_Line2 )
   END_RUNG
   // the same network as SCL:
   #oPLC_Aux.i_fCarrierGasSelected_Line2 := #ioPowder_Feeder_Unit_In_Out.Inputs.i_fCarrierGasSelected_Line2 AND "M_DUMMY_OFF";
END_REGION

REGION Network 39: HMI - CARRIER GAS SELECTED AUX
   RUNG wire#powerrail
      Contact( #oPLC_Aux.o_fCarrierGasSelect )
      Contact( "M_DUMMY_OFF" )
      Coil( #oPLC_Aux.i_fCarrierGasSelectedAux )
   END_RUNG
   // the same network as SCL:
   #oPLC_Aux.i_fCarrierGasSelectedAux := #oPLC_Aux.o_fCarrierGasSelect AND "M_DUMMY_OFF";
END_REGION

REGION Network 40: HMI - UNIT SELECTED LINE 1
   RUNG wire#powerrail
      Contact( #ioPowder_Feeder_Unit_In_Out.Inputs.i_fUnitSelected_Line1 )
      Coil( #oPLC_Aux.i_fUnitSelected_Line1 )
   END_RUNG
   // the same network as SCL:
   #oPLC_Aux.i_fUnitSelected_Line1 := #ioPowder_Feeder_Unit_In_Out.Inputs.i_fUnitSelected_Line1;
END_REGION

REGION Network 41: HMI - UNIT SELECTED LINE 2
   RUNG wire#powerrail
      Contact( #ioPowder_Feeder_Unit_In_Out.Inputs.i_fUnitSelected_Line2 )
      Coil( #oPLC_Aux.i_fUnitSelected_Line2 )
   END_RUNG
   // the same network as SCL:
   #oPLC_Aux.i_fUnitSelected_Line2 := #ioPowder_Feeder_Unit_In_Out.Inputs.i_fUnitSelected_Line2;
END_REGION

REGION Network 42: HMI - UNIT SELECTED AUX
   RUNG wire#powerrail
      Contact( #ioPowder_Feeder_Unit_In_Out.Inputs.i_fUnitSelected_Line1 )
      Contact( #ioPowder_Feeder_Unit_In_Out.Inputs.i_fUnitSelected_Line2 )
      Coil( #oPLC_Aux.i_fUnitSelectedAux )
   END_RUNG
   // the same network as SCL:
   #oPLC_Aux.i_fUnitSelectedAux := #ioPowder_Feeder_Unit_In_Out.Inputs.i_fUnitSelected_Line1 AND #ioPowder_Feeder_Unit_In_Out.Inputs.i_fUnitSelected_Line2;
END_REGION

REGION Network 43: HMI - CARRIERGAS ACTUAL LINE 1
   #oPLC_Aux.i_rCarriergasActual_Line1 := SWAP(#ioPowder_Feeder_Unit_In_Out.Inputs."Actual PF Values".i_rCarriergasActual_Line1);
END_REGION

REGION Network 44: HMI - CARRIERGAS ACTUAL LINE 2
   #oPLC_Aux.i_rCarriergasActual_Line2 := SWAP(#ioPowder_Feeder_Unit_In_Out.Inputs."Actual PF Values".i_rCarriergasActual_Line2);
END_REGION

REGION Network 45: HMI - DISK ACTUAL LINE 1
   #oPLC_Aux.i_rDiskActual_Line1 := SWAP(#ioPowder_Feeder_Unit_In_Out.Inputs."Actual PF Values".i_rDiskActual_Line1);
END_REGION

REGION Network 46: HMI - DISK ACTUAL LINE 2
   #oPLC_Aux.i_rDiskActual_Line2 := SWAP(#ioPowder_Feeder_Unit_In_Out.Inputs."Actual PF Values".i_rDiskActual_Line2);
END_REGION

REGION Network 47: HMI - STIRRER ACTUAL LINE 1
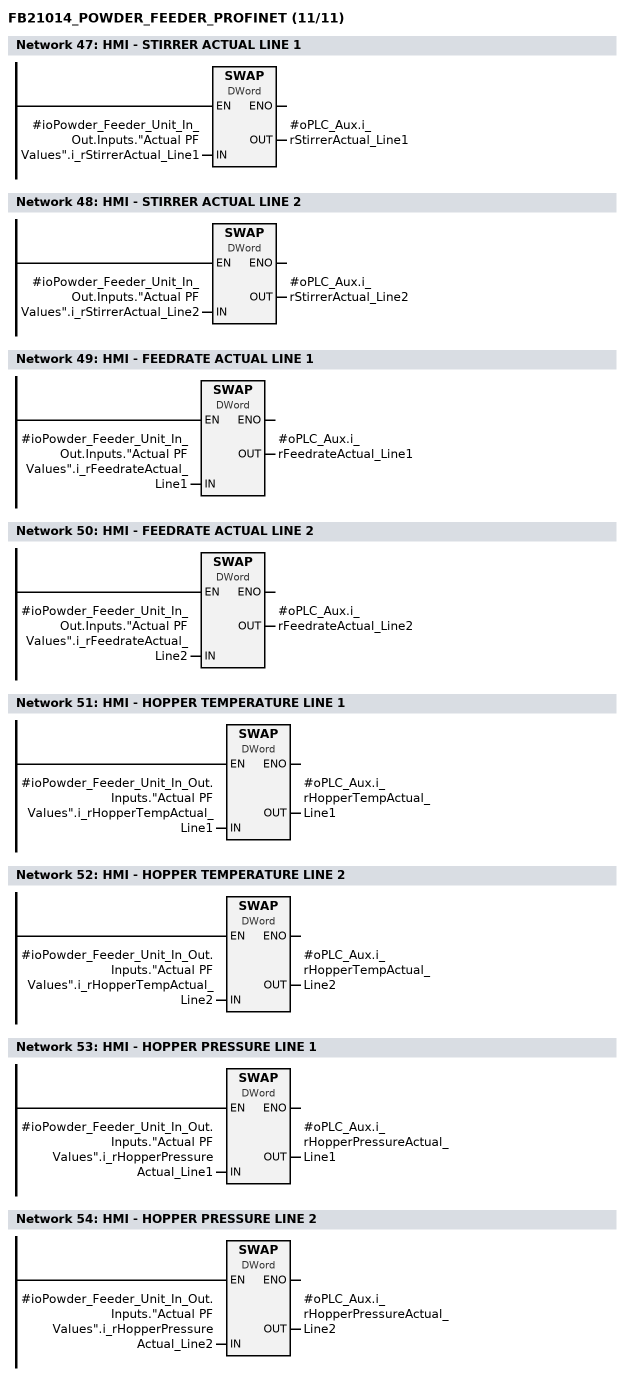
   #oPLC_Aux.i_rStirrerActual_Line1 := SWAP(#ioPowder_Feeder_Unit_In_Out.Inputs."Actual PF Values".i_rStirrerActual_Line1);
END_REGION

REGION Network 48: HMI - STIRRER ACTUAL LINE 2
   #oPLC_Aux.i_rStirrerActual_Line2 := SWAP(#ioPowder_Feeder_Unit_In_Out.Inputs."Actual PF Values".i_rStirrerActual_Line2);
END_REGION

REGION Network 49: HMI - FEEDRATE ACTUAL LINE 1
   #oPLC_Aux.i_rFeedrateActual_Line1 := SWAP(#ioPowder_Feeder_Unit_In_Out.Inputs."Actual PF Values".i_rFeedrateActual_Line1);
END_REGION

REGION Network 50: HMI - FEEDRATE ACTUAL LINE 2
   #oPLC_Aux.i_rFeedrateActual_Line2 := SWAP(#ioPowder_Feeder_Unit_In_Out.Inputs."Actual PF Values".i_rFeedrateActual_Line2);
END_REGION

REGION Network 51: HMI - HOPPER TEMPERATURE LINE 1
   #oPLC_Aux.i_rHopperTempActual_Line1 := SWAP(#ioPowder_Feeder_Unit_In_Out.Inputs."Actual PF Values".i_rHopperTempActual_Line1);
END_REGION

REGION Network 52: HMI - HOPPER TEMPERATURE LINE 2
   #oPLC_Aux.i_rHopperTempActual_Line2 := SWAP(#ioPowder_Feeder_Unit_In_Out.Inputs."Actual PF Values".i_rHopperTempActual_Line2);
END_REGION

REGION Network 53: HMI - HOPPER PRESSURE LINE 1
   #oPLC_Aux.i_rHopperPressureActual_Line1 := SWAP(#ioPowder_Feeder_Unit_In_Out.Inputs."Actual PF Values".i_rHopperPressureActual_Line1);
END_REGION

REGION Network 54: HMI - HOPPER PRESSURE LINE 2
   #oPLC_Aux.i_rHopperPressureActual_Line2 := SWAP(#ioPowder_Feeder_Unit_In_Out.Inputs."Actual PF Values".i_rHopperPressureActual_Line2);
END_REGION
END_FUNCTION_BLOCK
